EC00843=798156,1112951
EC00844=798156,1112951
EC00845=798156,1112951
EC00846=798156,1112951
EC00847=798156,1112951
EC00848=798156,1112951
EC00849=798156,1112951
EC00850=798156,1112951
EC00851=798156,1112951
EC00852=798156,1112951
EC00853=798156,1112951
EC00854=798156,1112951
EC00855=798156,1112951
EC00856=798156,1112951
EC00857=798156,1112951
EC00858=798156,1112951
EC00859=798156,1112951
EC00860=798156,1112951
EC00861=798156,1112951
EC00862=798156,1112951
EC00863=798156,1112951
EC00864=798156,1112951
EC00865=798156,1112951
EC00866=798156,1112951
EC00867=798156,1112951
EC00868=798156,1112951
EC00869=798156,1112951
EC00870=798156,1112951
EC00871=798156,1112951
EC00872=798156,1112951
EC00873=798156,1112951
EC00874=798156,1112951
EC00875=798156,1112951
EC00876=798156,1112951
EC00877=798156,1112949
EC00878=798156,1112951
EC00879=798156,1112951
EC00880=798156,1112951
EC00881=798156,1112951
EC00882=798156,1112951
EC00883=798156,1112951
EC00884=798156,1112951
EC00885=798156,1112951
EC00886=798156,1112951
EC00887=798156,1112951
EC00888=798156,1112951
EC00889=798156,1112951
EC00890=798156,1112951
EC00891=798156,1112951
EC00892=798156,1112951
EC00893=798156,1112951
EC00894=798156,1112951
EC00895=798156,1112951
EC00896=798156,1112951
EC00897=798156,1112951
EC00898=798156,1112951
EC00899=798156,1112951
EC00900=798156,1112951
EC00901=798156,1112951
EC00902=798156,1112951
EC00903=798156,1112951
EC00904=798156,1112951
EC00905=798156,1112951
EC00906=798156,1112951
EC00907=798156,1112951
EC00908=798156,1112951
EC00909=798156,1112951
EC00910=798156,1112951
EC00911=798156,1112951
EC00912=798156,1112951
EC00913=798156,1112951
EC00914=798156,1112951
EC00915=798156,1112951
EC00916=798156,1112951
EC00917=798156,1112951
EC00918=798156,1112951
EC00919=798156,1112951
EC00920=798156,1112951
EC00921=798156,1112951
EC00922=798156,1112951
EC00923=798156,1112951
EC00924=798156,1112951
EC00925=798156,1112951
EC00926=798156,1112951
EC00927=798156,1112951
EC00928=798156,1112951
EC00929=798156,1112951
EC00930=798156,1112951
EC00931=798156,1112951
EC00932=798156,1112951
EC00933=798156,1112951
EC00934=798156,1112951
EC00935=798156,1112951
EC00936=798156,1112951
EC00937=798156,1112951
EC00938=798156,1112951
EC00939=798156,1112951
EC00940=798156,1112951
EC00941=798156,1112951
EC00942=798155,1112950
EC00943=798155,1112950
EC00944=798155,1112950
EC00945=798155,1112950
EC00946=798155,1112950
EC00947=798155,1112950
EC00948=798155,1112950
EC00949=798156,1112951
EC00950=798156,1112951
EC00951=798156,1112951
EC00952=798156,1112951
EC00953=798156,1112951
EC00954=798156,1112951
EC00955=798156,1112951
EC00956=798156,1112951
EC00957=798156,1112951
EC00958=798156,1112951
EC00959=798156,1112951
EC00960=798156,1112951
EC00961=798156,1112951
EC00962=798156,1112951
EC00963=798156,1112951
EC00964=798156,1112951
EC00965=798156,1112951
EC00966=798156,1112951
EC00967=798156,1112951
EC00968=798156,1112951
EC00969=798156,1112951
EC00970=798156,1112951
EC00971=798156,1112951
EC00972=798156,1112951
EC00973=798156,1112951
EC00974=798156,1112951
EC00975=798156,1112951
EC00976=798156,1112951
EC00977=798156,1112951
EC00978=798156,1112951
EC00979=798156,1112951
EC00980=798156,1112951
EC00981=798156,1112951
EC00982=798156,1112951
EC00983=798156,1112951
EC00984=798156,1112951
EC00985=798156,1112951
EC00986=798156,1112951
EC00987=798156,1112951
EC00988=798156,1112951
EC00989=798156,1112951
EC00990=798156,1112951
EC00991=798156,1112951
EC00992=798156,1112951
EC00993=798156,1112951
EC00994=798156,1112951
EC00995=798156,1112951
EC00996=798156,1112951
EC00997=798156,1112951
EC00998=798156,1112951
EC00999=798156,1112951
EC01000=798156,1112951
EC01001=798156,1112951
EC01002=798156,1112951
EC01003=798156,1112951
EC01004=798156,1112951
EC01005=798156,1112951
EC01006=798156,1112951
EC01007=798156,1112951
EC01008=798156,1112951
EC01009=798156,1112951
EC01010=798156,1112951
EC01011=798156,1112951
EC01012=798156,1112951
EC01013=798156,1112951
EC01014=798156,1112951
EC01015=798156,1112951
EC01016=798155,1112949
EC01017=798156,1112951
EC01018=798156,1112951
EC01019=798156,1112951
EC01020=798156,1112951
EC01021=798156,1112951
EC01022=798156,1112951
EC01023=798156,1112951
EC01024=798156,1112951
EC01025=798156,1112951
EC01026=798156,1112951
EC01027=798156,1112951
EC01028=798156,1112951
EC01029=798156,1112951
EC01030=798156,1112951
EC01031=798156,1112951
EC01032=798156,1112951
EC01033=798156,1112951
EC01034=798156,1112951
///POSTYPE BASE
///RECTAN
///RCONF 0,0,0,0,0,0,0,0,0,0,0,0,0,0,0,0,0,0,0,0,0,0,0,0
P00006=0.222,-3.123,-1.508,0.0000,0.0000,0.0000
P00021=-0.225,-6.128,-0.405,0.0000,0.0000,0.0000
P00022=0.222,-3.123,-1.508,0.0000,0.0000,0.0000
P00023=0.143,-0.036,0.682,0.0000,0.0000,0.0000
P00024=0.145,-0.552,1.326,0.0000,0.0000,0.0000
P00025=-2.003,0.006,0.728,0.0000,0.0000,0.0000
P00026=0.562,-0.002,-0.337,0.0000,0.0000,0.0000
P00027=-0.746,0.015,-9.096,0.0000,0.0000,0.0000
P00028=-2.237,-0.018,-7.702,0.0000,0.0000,0.0000
P00029=-2.156,-0.086,-4.681,0.0000,0.0000,0.0000
P00030=5.926,-4.294,-1.390,0.0000,0.0000,0.0000
P00031=1.853,-0.001,-1.549,0.0000,0.0000,0.0000
P00032=1.957,0.503,-7.217,0.0000,0.0000,0.0000
///RCONF 0,0,0,0,1,0,0,0,0,0,0,0,0,0,0,0,0,0,0,0,0,0,0,0
P00033=-0.123,0.612,-5.012,0.0000,0.0000,0.0000
///RCONF 0,0,0,0,0,0,0,0,0,0,0,0,0,0,0,0,0,0,0,0,0,0,0,0
P00034=-0.304,0.773,-2.693,0.0000,0.0000,0.0000
P00035=2.817,0.591,-1.622,0.0000,0.0000,0.0000
P00040=-0.030,9.648,2.467,0.0000,0.0000,0.0000
P00041=0.192,3.924,0.305,0.0000,0.0000,0.0000
P00042=-0.217,1.941,0.413,0.0000,0.0000,0.0000
P00043=-0.044,-1.937,1.197,0.0000,0.0000,0.0000
P00044=0.687,-2.322,1.156,0.0000,0.0000,0.0000
P00045=-0.068,-0.810,1.603,0.0000,0.0000,0.0000
P00046=0.799,0.043,1.292,0.0000,0.0000,0.0000
///RCONF 0,1,0,0,0,0,0,0,0,0,0,0,0,0,0,0,0,0,0,0,0,0,0,0
P00047=-0.011,1.737,-0.646,0.0000,0.0000,0.0000
///RCONF 0,0,0,0,0,0,0,0,0,0,0,0,0,0,0,0,0,0,0,0,0,0,0,0
P00048=2.411,0.025,-0.606,0.0000,0.0000,0.0000
P00049=3.413,-3.572,-1.618,0.0000,0.0000,0.0000
P00050=4.296,-4.501,-0.826,0.0000,0.0000,0.0000
P00051=0.367,3.892,0.009,0.0000,0.0000,0.0000
P00052=0.088,2.832,-0.342,0.0000,0.0000,0.0000
P00053=0.134,6.594,0.107,0.0000,0.0000,0.0000
P00054=-0.103,6.509,-0.702,0.0000,0.0000,0.0000
P00061=1.575,-3.405,-0.752,0.0000,0.0000,0.0000
P00062=-0.135,-0.848,-1.706,0.0000,0.0000,0.0000
P00063=0.036,-0.654,-3.005,0.0000,0.0000,0.0000
P00071=2.716,0.070,1.352,0.0000,0.0000,0.0000
P00072=1.041,-0.003,-0.797,0.0000,0.0000,0.0000
P00073=-0.961,5.319,-6.157,0.0000,0.0000,0.0000
P00074=1.123,1.944,-5.914,0.0000,0.0000,0.0000
P00080=-3.893,-3.240,-0.208,0.0000,0.0000,0.0000
P00081=19.486,11.347,1.262,0.0000,0.0000,0.0000
P00088=-2.376,0.094,2.453,0.0000,0.0000,0.0000
P00089=5.697,-3.100,-1.263,0.0000,0.0000,0.0000
P00095=-3.945,4.918,-0.177,0.0000,0.0000,0.0000
P00096=-0.633,5.398,-3.809,0.0000,0.0000,0.0000
//INST
///DATE 2024/08/30 11:58
///ATTR SC,RW
///GROUP1 RB1,BS1
///GROUP2 ST1
NOP
'X2_8B-21B(90,180)
'
MOVJ C00000 BC00000 VJ=100.00  +MOVJ EC00000 VJ=100.00
'Path S4722
SFTOF3D
MOVJ C00001 BC00001 VJ=100.00  +MOVJ EC00001 VJ=100.00
MOVL C00002 BC00002 V=666.7  +MOVJ EC00002 VJ=100.00
SMOVL C00003 BC00003 V=166.7  +MOVJ EC00003
SREFP 3 C00004 BC00004  +REFP EC00004
CALL JOB:SEARCH-R1-S13D
SET P095 P006
SFTON3D P095
SMOVL C00005 BC00005 V=166.7  +MOVJ EC00005
SREFP 3 C00006 BC00006  +REFP EC00006
CALL JOB:SEARCH-R1-S13D
SET P095 P006
SFTON3D P095
SMOVL C00007 BC00007 V=166.7  +MOVJ EC00007
MOVL C00008 BC00008 V=1000.0  +MOVJ EC00008 VJ=100.00
'EndPath S4722
'Path S4723
SFTOF3D
MOVJ C00009 BC00009 VJ=100.00  +MOVJ EC00009 VJ=100.00
MOVL C00010 BC00010 V=666.7  +MOVJ EC00010 VJ=100.00
SMOVL C00011 BC00011 V=166.7  +MOVJ EC00011
SREFP 3 C00012 BC00012  +REFP EC00012
CALL JOB:SEARCH-R1-S13D
SET P096 P006
SFTON3D P096
SMOVL C00013 BC00013 V=166.7  +MOVJ EC00013
SREFP 3 C00014 BC00014  +REFP EC00014
CALL JOB:SEARCH-R1-S13D
SET P096 P006
SFTON3D P096
SMOVL C00015 BC00015 V=166.7  +MOVJ EC00015
MOVL C00016 BC00016 V=1000.0  +MOVJ EC00016 VJ=100.00
'EndPath S4723
'
'
'Path S4093
SFTOF3D
MOVJ C00017 BC00017 VJ=100.00  +MOVJ EC00017 VJ=100.00
MOVL C00018 BC00018 V=666.7  +MOVJ EC00018 VJ=100.00
SMOVL C00019 BC00019 V=166.7  +MOVJ EC00019
SREFP 3 C00020 BC00020  +REFP EC00020
CALL JOB:SEARCH-R1-S13D
SET P021 P006
SFTON3D P021
SMOVL C00021 BC00021 V=166.7  +MOVJ EC00021
SREFP 3 C00022 BC00022  +REFP EC00022
CALL JOB:SEARCH-R1-S13D
SET P021 P006
SFTON3D P021
SMOVL C00023 BC00023 V=166.7  +MOVJ EC00023
MOVL C00024 BC00024 V=1000.0  +MOVJ EC00024 VJ=100.00
'EndPath S4093
'Path S4094
SFTOF3D
MOVJ C00025 BC00025 VJ=100.00  +MOVJ EC00025 VJ=100.00
MOVL C00026 BC00026 V=666.7  +MOVJ EC00026 VJ=100.00
SMOVL C00027 BC00027 V=166.7  +MOVJ EC00027
SREFP 3 C00028 BC00028  +REFP EC00028
CALL JOB:SEARCH-R1-S13D
SET P022 P006
SFTON3D P022
SMOVL C00029 BC00029 V=166.7  +MOVJ EC00029
SREFP 3 C00030 BC00030  +REFP EC00030
CALL JOB:SEARCH-R1-S13D
SET P022 P006
SFTON3D P022
SMOVL C00031 BC00031 V=166.7  +MOVJ EC00031
MOVL C00032 BC00032 V=1000.0  +MOVJ EC00032 VJ=100.00
'EndPath S4094
MOVJ C00033 BC00033 VJ=100.00  +MOVJ EC00033 VJ=100.00
'Path S4205
SFTOF3D
MOVJ C00034 BC00034 VJ=100.00  +MOVJ EC00034 VJ=100.00
MOVL C00035 BC00035 V=666.7  +MOVJ EC00035 VJ=100.00
SMOVL C00036 BC00036 V=166.7  +MOVJ EC00036
SREFP 3 C00037 BC00037  +REFP EC00037
CALL JOB:SEARCH-R1-S13D
SET P050 P006
SFTON3D P050
SMOVL C00038 BC00038 V=166.7  +MOVJ EC00038
SREFP 3 C00039 BC00039  +REFP EC00039
CALL JOB:SEARCH-R1-S13D
SET P050 P006
SFTON3D P050
SMOVL C00040 BC00040 V=166.7  +MOVJ EC00040
SMOVL C00041 BC00041 V=250.0  +MOVJ EC00041
SMOVL C00042 BC00042 V=166.7  +MOVJ EC00042
SREFP 3 C00043 BC00043  +REFP EC00043
CALL JOB:SEARCH-R1-S13D
SET P050 P006
SFTON3D P050
SMOVL C00044 BC00044 V=250.0  +MOVJ EC00044
'EndPath S4205
'Path S4206
SFTOF3D
MOVL C00045 BC00045 V=1000.0  +MOVJ EC00045 VJ=100.00
SMOVL C00046 BC00046 V=166.7  +MOVJ EC00046
SREFP 3 C00047 BC00047  +REFP EC00047
CALL JOB:SEARCH-R1-S13D
SET P051 P006
SFTON3D P051
SMOVL C00048 BC00048 V=166.7  +MOVJ EC00048
SREFP 3 C00049 BC00049  +REFP EC00049
CALL JOB:SEARCH-R1-S13D
SET P051 P006
SFTON3D P051
SMOVL C00050 BC00050 V=166.7  +MOVJ EC00050
SMOVL C00051 BC00051 V=250.0  +MOVJ EC00051
SREFP 3 C00052 BC00052  +REFP EC00052
CALL JOB:SEARCH-R1-S13D
SET P051 P006
SFTON3D P051
SMOVL C00053 BC00053 V=250.0  +MOVJ EC00053
MOVL C00054 BC00054 V=1000.0  +MOVJ EC00054 VJ=100.00
'EndPath S4206
MOVJ C00055 BC00055 VJ=100.00  +MOVJ EC00055 VJ=100.00
'Path S4207
SFTOF3D
MOVJ C00056 BC00056 VJ=100.00  +MOVJ EC00056 VJ=100.00
MOVL C00057 BC00057 V=666.7  +MOVJ EC00057 VJ=100.00
SMOVL C00058 BC00058 V=166.7  +MOVJ EC00058
SREFP 3 C00059 BC00059  +REFP EC00059
CALL JOB:SEARCH-R1-S13D
SET P054 P006
SFTON3D P054
SMOVL C00060 BC00060 V=250.0  +MOVJ EC00060
SMOVL C00061 BC00061 V=233.3  +MOVJ EC00061
SMOVL C00062 BC00062 V=166.7  +MOVJ EC00062
SREFP 3 C00063 BC00063  +REFP EC00063
CALL JOB:SEARCH-R1-S13D
SET P054 P006
SFTON3D P054
SMOVL C00064 BC00064 V=166.7  +MOVJ EC00064
SMOVL C00065 BC00065 V=416.7  +MOVJ EC00065
SMOVL C00066 BC00066 V=250.0  +MOVJ EC00066
SREFP 3 C00067 BC00067  +REFP EC00067
CALL JOB:SEARCH-R1-S13D
SET P054 P006
SFTON3D P054
SMOVL C00068 BC00068 V=250.0  +MOVJ EC00068
MOVL C00069 BC00069 V=1000.0  +MOVJ EC00069 VJ=100.00
'EndPath S4207
'Path S4095
SFTOF3D
MOVJ C00070 BC00070 VJ=100.00  +MOVJ EC00070 VJ=100.00
MOVJ C00071 BC00071 VJ=100.00  +MOVJ EC00071 VJ=100.00
SMOVL C00072 BC00072 V=200.0  +MOVJ EC00072
SREFP 3 C00073 BC00073  +REFP EC00073
CALL JOB:SEARCH-R1-S13D
SET P089 P006
SFTON3D P089
SMOVL C00074 BC00074 V=166.7  +MOVJ EC00074
SMOVL C00075 BC00075 V=166.7  +MOVJ EC00075
SREFP 3 C00076 BC00076  +REFP EC00076
CALL JOB:SEARCH-R1-S13D
SET P089 P006
SFTON3D P089
SMOVL C00077 BC00077 V=166.7  +MOVJ EC00077
SMOVL C00078 BC00078 V=166.7  +MOVJ EC00078
SREFP 3 C00079 BC00079  +REFP EC00079
CALL JOB:SEARCH-R1-S13D
SET P089 P006
SFTON3D P089
SMOVL C00080 BC00080 V=166.7  +MOVJ EC00080
SMOVL C00081 BC00081 V=1000.0  +MOVJ EC00081
SFTOF3D
MOVJ C00082 BC00082 VJ=100.00  +MOVJ EC00082 VJ=100.00
MOVL C00083 BC00083 V=666.7  +MOVJ EC00083 VJ=100.00
SMOVL C00084 BC00084 V=166.7  +MOVJ EC00084
SREFP 3 C00085 BC00085  +REFP EC00085
CALL JOB:SEARCH-R1-S13D
SET P034 P006
SFTON3D P034
SMOVL C00086 BC00086 V=250.0  +MOVJ EC00086
SMOVL C00087 BC00087 V=233.3  +MOVJ EC00087
SMOVL C00088 BC00088 V=166.7  +MOVJ EC00088
SREFP 3 C00089 BC00089  +REFP EC00089
CALL JOB:SEARCH-R1-S13D
SET P034 P006
SFTON3D P034
SMOVL C00090 BC00090 V=166.7  +MOVJ EC00090
SMOVL C00091 BC00091 V=166.7  +MOVJ EC00091
SREFP 3 C00092 BC00092  +REFP EC00092
CALL JOB:SEARCH-R1-S13D
SET P034 P006
SFTON3D P034
SMOVL C00093 BC00093 V=166.7  +MOVJ EC00093
MOVJ C00094 BC00094 VJ=50.00  +MOVJ EC00094 VJ=30.00
'EndPath S4095
'Path S4096
SFTOF3D
MOVJ C00095 BC00095 VJ=50.00  +MOVJ EC00095 VJ=30.00
MOVJ C00096 BC00096 VJ=50.00  +MOVJ EC00096 VJ=30.00
MOVJ C00097 BC00097 VJ=50.00  +MOVJ EC00097 VJ=30.00
SMOVL C00098 BC00098 V=166.7  +MOVJ EC00098
SREFP 3 C00099 BC00099  +REFP EC00099
CALL JOB:SEARCH-R1-S13D
SET P061 P006
SFTON3D P061
SMOVL C00100 BC00100 V=166.7  +MOVJ EC00100
SREFP 3 C00101 BC00101  +REFP EC00101
CALL JOB:SEARCH-R1-S13D
SET P061 P006
SFTON3D P061
SMOVL C00102 BC00102 V=166.7  +MOVJ EC00102
SFTOF3D
SMOVL C00103 BC00103 V=666.7  +MOVJ EC00103
SMOVL C00104 BC00104 V=166.7  +MOVJ EC00104
SREFP 3 C00105 BC00105  +REFP EC00105
CALL JOB:SEARCH-R1-S13D
SET P062 P006
SFTON3D P062
SMOVL C00106 BC00106 V=166.7  +MOVJ EC00106
SREFP 3 C00107 BC00107  +REFP EC00107
CALL JOB:SEARCH-R1-S13D
SET P062 P006
SFTON3D P062
SMOVL C00108 BC00108 V=250.0  +MOVJ EC00108
SFTOF3D
SMOVL C00109 BC00109 V=500.0  +MOVJ EC00109
SMOVL C00110 BC00110 V=166.7  +MOVJ EC00110
SREFP 3 C00111 BC00111  +REFP EC00111
CALL JOB:SEARCH-R1-S13D
SET P063 P006
SFTON3D P063
SMOVL C00112 BC00112 V=166.7  +MOVJ EC00112
SREFP 3 C00113 BC00113  +REFP EC00113
CALL JOB:SEARCH-R1-S13D
SET P063 P006
SFTON3D P063
SMOVL C00114 BC00114 V=166.7  +MOVJ EC00114
SFTOF3D
SMOVL C00115 BC00115 V=1000.0  +MOVJ EC00115
MOVJ C00116 BC00116 VJ=100.00  +MOVJ EC00116 VJ=30.00
MOVJ C00117 BC00117 VJ=50.00  +MOVJ EC00117 VJ=30.00
MOVJ C00118 BC00118 VJ=100.00  +MOVJ EC00118 VJ=100.00
MOVL C00119 BC00119 V=666.7  +MOVJ EC00119 VJ=100.00
SMOVL C00120 BC00120 V=166.7  +MOVJ EC00120
SREFP 3 C00121 BC00121  +REFP EC00121
CALL JOB:SEARCH-R1-S13D
SET P023 P006
SFTON3D P023
SMOVL C00122 BC00122 V=166.7  +MOVJ EC00122
SMOVL C00123 BC00123 V=333.3  +MOVJ EC00123
SMOVL C00124 BC00124 V=166.7  +MOVJ EC00124
SREFP 3 C00125 BC00125  +REFP EC00125
CALL JOB:SEARCH-R1-S13D
SET P023 P006
SFTON3D P023
SMOVL C00126 BC00126 V=166.7  +MOVJ EC00126
SMOVL C00127 BC00127 V=166.7  +MOVJ EC00127
SREFP 3 C00128 BC00128  +REFP EC00128
CALL JOB:SEARCH-R1-S13D
SET P023 P006
SFTON3D P023
SMOVL C00129 BC00129 V=166.7  +MOVJ EC00129
MOVL C00130 BC00130 V=1000.0  +MOVJ EC00130 VJ=100.00
'EndPath S4096
MOVJ C00131 BC00131 VJ=100.00  +MOVJ EC00131 VJ=100.00
'Path S4097
SFTOF3D
MOVJ C00132 BC00132 VJ=100.00  +MOVJ EC00132 VJ=100.00
MOVL C00133 BC00133 V=666.7  +MOVJ EC00133 VJ=100.00
SMOVL C00134 BC00134 V=166.7  +MOVJ EC00134
SREFP 3 C00135 BC00135  +REFP EC00135
CALL JOB:SEARCH-R1-S13D
SET P024 P006
SFTON3D P024
SMOVL C00136 BC00136 V=166.7  +MOVJ EC00136
SREFP 3 C00137 BC00137  +REFP EC00137
CALL JOB:SEARCH-R1-S13D
SET P024 P006
SFTON3D P024
SMOVL C00138 BC00138 V=166.7  +MOVJ EC00138
SMOVL C00139 BC00139 V=166.7  +MOVJ EC00139
SREFP 3 C00140 BC00140  +REFP EC00140
CALL JOB:SEARCH-R1-S13D
SET P024 P006
SFTON3D P024
SMOVL C00141 BC00141 V=166.7  +MOVJ EC00141
MOVL C00142 BC00142 V=1000.0  +MOVJ EC00142 VJ=100.00
'EndPath S4097
'Path S4098
SFTOF3D
MOVJ C00143 BC00143 VJ=100.00  +MOVJ EC00143 VJ=100.00
MOVL C00144 BC00144 V=666.7  +MOVJ EC00144 VJ=100.00
SMOVL C00145 BC00145 V=166.7  +MOVJ EC00145
SREFP 3 C00146 BC00146  +REFP EC00146
CALL JOB:SEARCH-R1-S13D
SET P035 P006
SFTON3D P035
SMOVL C00147 BC00147 V=166.7  +MOVJ EC00147
SREFP 3 C00148 BC00148  +REFP EC00148
CALL JOB:SEARCH-R1-S13D
SET P035 P006
SFTON3D P035
SMOVL C00149 BC00149 V=166.7  +MOVJ EC00149
SMOVL C00150 BC00150 V=166.7  +MOVJ EC00150
SMOVL C00151 BC00151 V=166.7  +MOVJ EC00151
SREFP 3 C00152 BC00152  +REFP EC00152
CALL JOB:SEARCH-R1-S13D
SET P035 P006
SFTON3D P035
SMOVL C00153 BC00153 V=166.7  +MOVJ EC00153
MOVL C00154 BC00154 V=1000.0  +MOVJ EC00154 VJ=100.00
'EndPath S4098
'Path S4099
SFTOF3D
MOVJ C00155 BC00155 VJ=100.00  +MOVJ EC00155 VJ=100.00
MOVL C00156 BC00156 V=666.7  +MOVJ EC00156 VJ=100.00
SMOVL C00157 BC00157 V=166.7  +MOVJ EC00157
SREFP 3 C00158 BC00158  +REFP EC00158
CALL JOB:SEARCH-R1-S13D
SET P029 P006
SFTON3D P029
SMOVL C00159 BC00159 V=166.7  +MOVJ EC00159
SREFP 3 C00160 BC00160  +REFP EC00160
CALL JOB:SEARCH-R1-S13D
SET P029 P006
SFTON3D P029
SMOVL C00161 BC00161 V=166.7  +MOVJ EC00161
SMOVL C00162 BC00162 V=250.0  +MOVJ EC00162
SMOVL C00163 BC00163 V=166.7  +MOVJ EC00163
SREFP 3 C00164 BC00164  +REFP EC00164
CALL JOB:SEARCH-R1-S13D
SET P029 P006
SFTON3D P029
SMOVL C00165 BC00165 V=166.7  +MOVJ EC00165
'EndPath S4099
'Path S4855
SFTOF3D
MOVL C00166 BC00166 V=666.7  +MOVJ EC00166 VJ=100.00
SMOVL C00167 BC00167 V=166.7  +MOVJ EC00167
SREFP 3 C00168 BC00168  +REFP EC00168
CALL JOB:SEARCH-R1-S13D
SET P071 P006
SFTON3D P071
SMOVL C00169 BC00169 V=166.7  +MOVJ EC00169
SREFP 3 C00170 BC00170  +REFP EC00170
CALL JOB:SEARCH-R1-S13D
SET P071 P006
SFTON3D P071
SMOVL C00171 BC00171 V=166.7  +MOVJ EC00171
SMOVL C00172 BC00172 V=166.7  +MOVJ EC00172
SREFP 3 C00173 BC00173  +REFP EC00173
CALL JOB:SEARCH-R1-S13D
SET P071 P006
SFTON3D P071
SMOVL C00174 BC00174 V=166.7  +MOVJ EC00174
MOVL C00175 BC00175 V=1000.0  +MOVJ EC00175 VJ=100.00
MOVL C00176 BC00176 V=666.7  +MOVJ EC00176 VJ=100.00
SMOVL C00177 BC00177 V=166.7  +MOVJ EC00177
SREFP 3 C00178 BC00178  +REFP EC00178
CALL JOB:SEARCH-R1-S13D
SET P080 P006
SFTON3D P080
SMOVL C00179 BC00179 V=166.7  +MOVJ EC00179
SREFP 3 C00180 BC00180  +REFP EC00180
CALL JOB:SEARCH-R1-S13D
SET P080 P006
SFTON3D P080
SMOVL C00181 BC00181 V=166.7  +MOVJ EC00181
SMOVL C00182 BC00182 V=250.0  +MOVJ EC00182
SMOVL C00183 BC00183 V=166.7  +MOVJ EC00183
SREFP 3 C00184 BC00184  +REFP EC00184
CALL JOB:SEARCH-R1-S13D
SET P080 P006
SFTON3D P080
SMOVL C00185 BC00185 V=166.7  +MOVJ EC00185
'EndPath S4855
'Path S4856
SFTOF3D
MOVJ C00186 BC00186 VJ=100.00  +MOVJ EC00186 VJ=100.00
MOVL C00187 BC00187 V=666.7  +MOVJ EC00187 VJ=100.00
SMOVL C00188 BC00188 V=166.7  +MOVJ EC00188
SREFP 3 C00189 BC00189  +REFP EC00189
CALL JOB:SEARCH-R1-S13D
SET P072 P006
SFTON3D P072
SMOVL C00190 BC00190 V=166.7  +MOVJ EC00190
SREFP 3 C00191 BC00191  +REFP EC00191
CALL JOB:SEARCH-R1-S13D
SET P072 P006
SFTON3D P072
SMOVL C00192 BC00192 V=166.7  +MOVJ EC00192
MOVL C00193 BC00193 V=1000.0  +MOVJ EC00193 VJ=100.00
'EndPath S4856
MOVJ C00194 BC00194 VJ=100.00  +MOVJ EC00194 VJ=100.00
'Path S4857
SFTOF3D
MOVJ C00195 BC00195 VJ=100.00  +MOVJ EC00195 VJ=100.00
MOVL C00196 BC00196 V=666.7  +MOVJ EC00196 VJ=100.00
SMOVL C00197 BC00197 V=166.7  +MOVJ EC00197
SREFP 3 C00198 BC00198  +REFP EC00198
CALL JOB:SEARCH-R1-S13D
SET P073 P006
SFTON3D P073
SMOVL C00199 BC00199 V=166.7  +MOVJ EC00199
SMOVL C00200 BC00200 V=166.7  +MOVJ EC00200
SREFP 3 C00201 BC00201  +REFP EC00201
CALL JOB:SEARCH-R1-S13D
SET P073 P006
SFTON3D P073
SMOVL C00202 BC00202 V=166.7  +MOVJ EC00202
SMOVL C00203 BC00203 V=166.7  +MOVJ EC00203
SREFP 3 C00204 BC00204  +REFP EC00204
CALL JOB:SEARCH-R1-S13D
SET P073 P006
SFTON3D P073
SMOVL C00205 BC00205 V=166.7  +MOVJ EC00205
MOVL C00206 BC00206 V=1000.0  +MOVJ EC00206 VJ=100.00
'EndPath S4857
MOVJ C00207 BC00207 VJ=100.00  +MOVJ EC00207 VJ=100.00
MOVJ C00208 BC00208 VJ=100.00  +MOVJ EC00208 VJ=100.00
'Path S4858
SFTOF3D
MOVJ C00209 BC00209 VJ=100.00  +MOVJ EC00209 VJ=100.00
MOVL C00210 BC00210 V=666.7  +MOVJ EC00210 VJ=100.00
SMOVL C00211 BC00211 V=166.7  +MOVJ EC00211
SREFP 3 C00212 BC00212  +REFP EC00212
CALL JOB:SEARCH-R1-S13D
SET P074 P006
SFTON3D P074
SMOVL C00213 BC00213 V=166.7  +MOVJ EC00213
SREFP 3 C00214 BC00214  +REFP EC00214
CALL JOB:SEARCH-R1-S13D
SET P074 P006
SFTON3D P074
SMOVL C00215 BC00215 V=166.7  +MOVJ EC00215
MOVL C00216 BC00216 V=1000.0  +MOVJ EC00216 VJ=100.00
'EndPath S4858
MOVJ C00217 BC00217 VJ=100.00  +MOVJ EC00217 VJ=100.00
MOVJ C00218 BC00218 VJ=100.00  +MOVJ EC00218 VJ=100.00
'Path S4100
SFTOF3D
MOVJ C00219 BC00219 VJ=100.00  +MOVJ EC00219 VJ=100.00
MOVL C00220 BC00220 V=666.7  +MOVJ EC00220 VJ=100.00
SMOVL C00221 BC00221 V=166.7  +MOVJ EC00221
SREFP 3 C00222 BC00222  +REFP EC00222
CALL JOB:SEARCH-R1-S13D
SET P081 P006
SFTON3D P081
SMOVL C00223 BC00223 V=166.7  +MOVJ EC00223
SREFP 3 C00224 BC00224  +REFP EC00224
CALL JOB:SEARCH-R1-S13D
SET P081 P006
SFTON3D P081
SMOVL C00225 BC00225 V=166.7  +MOVJ EC00225
SMOVL C00226 BC00226 V=666.7  +MOVJ EC00226
SMOVL C00227 BC00227 V=666.7  +MOVJ EC00227
SMOVL C00228 BC00228 V=666.7  +MOVJ EC00228
SMOVL C00229 BC00229 V=166.7  +MOVJ EC00229
SREFP 3 C00230 BC00230  +REFP EC00230
CALL JOB:SEARCH-R1-S13D
SET P081 P006
SFTON3D P081
SMOVL C00231 BC00231 V=250.0  +MOVJ EC00231
SMOVL C00232 BC00232 V=666.7  +MOVJ EC00232
MOVJ C00233 BC00233 VJ=100.00  +MOVJ EC00233 VJ=100.00
MOVL C00234 BC00234 V=666.7  +MOVJ EC00234 VJ=100.00
SMOVL C00235 BC00235 V=166.7  +MOVJ EC00235
SREFP 3 C00236 BC00236  +REFP EC00236
CALL JOB:SEARCH-R1-S13D
SET P026 P006
SFTON3D P026
SMOVL C00237 BC00237 V=166.7  +MOVJ EC00237
SREFP 3 C00238 BC00238  +REFP EC00238
CALL JOB:SEARCH-R1-S13D
SET P026 P006
SFTON3D P026
SMOVL C00239 BC00239 V=166.7  +MOVJ EC00239
SMOVL C00240 BC00240 V=666.7  +MOVJ EC00240
SMOVL C00241 BC00241 V=666.7  +MOVJ EC00241
SMOVL C00242 BC00242 V=666.7  +MOVJ EC00242
SMOVL C00243 BC00243 V=166.7  +MOVJ EC00243
SREFP 3 C00244 BC00244  +REFP EC00244
CALL JOB:SEARCH-R1-S13D
SET P026 P006
SFTON3D P026
SMOVL C00245 BC00245 V=250.0  +MOVJ EC00245
SMOVL C00246 BC00246 V=666.7  +MOVJ EC00246
MOVL C00247 BC00247 V=1000.0  +MOVJ EC00247 VJ=100.00
'EndPath S4100
MOVJ C00248 BC00248 VJ=50.00  +MOVJ EC00248 VJ=100.00
'Path S4101
SFTOF3D
MOVJ C00249 BC00249 VJ=50.00  +MOVJ EC00249 VJ=100.00
MOVL C00250 BC00250 V=666.7  +MOVJ EC00250 VJ=100.00
SMOVL C00251 BC00251 V=166.7  +MOVJ EC00251
SREFP 3 C00252 BC00252  +REFP EC00252
CALL JOB:SEARCH-R1-S13D
SET P025 P006
SFTON3D P025
SMOVL C00253 BC00253 V=166.7  +MOVJ EC00253
SREFP 3 C00254 BC00254  +REFP EC00254
CALL JOB:SEARCH-R1-S13D
SET P025 P006
SFTON3D P025
SMOVL C00255 BC00255 V=166.7  +MOVJ EC00255
SMOVL C00256 BC00256 V=333.3  +MOVJ EC00256
SMOVL C00257 BC00257 V=166.7  +MOVJ EC00257
SREFP 3 C00258 BC00258  +REFP EC00258
CALL JOB:SEARCH-R1-S13D
SET P025 P006
SFTON3D P025
SMOVL C00259 BC00259 V=166.7  +MOVJ EC00259
MOVL C00260 BC00260 V=1000.0  +MOVJ EC00260 VJ=100.00
'EndPath S4101
MOVJ C00261 BC00261 VJ=100.00  +MOVJ EC00261 VJ=100.00
'Path S4102
SFTOF3D
MOVJ C00262 BC00262 VJ=100.00  +MOVJ EC00262 VJ=100.00
MOVL C00263 BC00263 V=666.7  +MOVJ EC00263 VJ=100.00
SMOVL C00264 BC00264 V=166.7  +MOVJ EC00264
SREFP 3 C00265 BC00265  +REFP EC00265
CALL JOB:SEARCH-R1-S13D
SET P028 P006
SFTON3D P028
SMOVL C00266 BC00266 V=166.7  +MOVJ EC00266
SREFP 3 C00267 BC00267  +REFP EC00267
CALL JOB:SEARCH-R1-S13D
SET P028 P006
SFTON3D P028
SMOVL C00268 BC00268 V=166.7  +MOVJ EC00268
SMOVL C00269 BC00269 V=333.3  +MOVJ EC00269
SMOVL C00270 BC00270 V=166.7  +MOVJ EC00270
SREFP 3 C00271 BC00271  +REFP EC00271
CALL JOB:SEARCH-R1-S13D
SET P028 P006
SFTON3D P028
SMOVL C00272 BC00272 V=166.7  +MOVJ EC00272
MOVL C00273 BC00273 V=1000.0  +MOVJ EC00273 VJ=100.00
'EndPath S4102
MOVJ C00274 BC00274 VJ=100.00  +MOVJ EC00274 VJ=100.00
'Path S4103
SFTOF3D
MOVJ C00275 BC00275 VJ=100.00  +MOVJ EC00275 VJ=100.00
MOVL C00276 BC00276 V=666.7  +MOVJ EC00276 VJ=100.00
SMOVL C00277 BC00277 V=166.7  +MOVJ EC00277
SREFP 3 C00278 BC00278  +REFP EC00278
CALL JOB:SEARCH-R1-S13D
SET P033 P006
SFTON3D P033
SMOVL C00279 BC00279 V=166.7  +MOVJ EC00279
SMOVL C00280 BC00280 V=166.7  +MOVJ EC00280
SREFP 3 C00281 BC00281  +REFP EC00281
CALL JOB:SEARCH-R1-S13D
SET P033 P006
SFTON3D P033
SMOVL C00282 BC00282 V=166.7  +MOVJ EC00282
SMOVL C00283 BC00283 V=166.7  +MOVJ EC00283
SMOVL C00284 BC00284 V=166.7  +MOVJ EC00284
SREFP 3 C00285 BC00285  +REFP EC00285
CALL JOB:SEARCH-R1-S13D
SET P033 P006
SFTON3D P033
SMOVL C00286 BC00286 V=166.7  +MOVJ EC00286
MOVL C00287 BC00287 V=1000.0  +MOVJ EC00287 VJ=100.00
'EndPath S4103
'Path S4104
SFTOF3D
MOVJ C00288 BC00288 VJ=100.00  +MOVJ EC00288 VJ=100.00
MOVL C00289 BC00289 V=666.7  +MOVJ EC00289 VJ=100.00
SMOVL C00290 BC00290 V=166.7  +MOVJ EC00290
SREFP 3 C00291 BC00291  +REFP EC00291
CALL JOB:SEARCH-R1-S13D
SET P027 P006
SFTON3D P027
SMOVL C00292 BC00292 V=250.0  +MOVJ EC00292
SMOVL C00293 BC00293 V=166.7  +MOVJ EC00293
SREFP 3 C00294 BC00294  +REFP EC00294
CALL JOB:SEARCH-R1-S13D
SET P027 P006
SFTON3D P027
SMOVL C00295 BC00295 V=166.7  +MOVJ EC00295
SMOVL C00296 BC00296 V=166.7  +MOVJ EC00296
SREFP 3 C00297 BC00297  +REFP EC00297
CALL JOB:SEARCH-R1-S13D
SET P027 P006
SFTON3D P027
SMOVL C00298 BC00298 V=166.7  +MOVJ EC00298
MOVL C00299 BC00299 V=1000.0  +MOVJ EC00299 VJ=100.00
'EndPath S4104
MOVJ C00300 BC00300 VJ=100.00  +MOVJ EC00300 VJ=100.00
'Path S4105
SFTOF3D
MOVJ C00301 BC00301 VJ=100.00  +MOVJ EC00301 VJ=100.00
MOVL C00302 BC00302 V=666.7  +MOVJ EC00302 VJ=100.00
SMOVL C00303 BC00303 V=166.7  +MOVJ EC00303
SREFP 3 C00304 BC00304  +REFP EC00304
CALL JOB:SEARCH-R1-S13D
SET P030 P006
SFTON3D P030
SMOVL C00305 BC00305 V=166.7  +MOVJ EC00305
SREFP 3 C00306 BC00306  +REFP EC00306
CALL JOB:SEARCH-R1-S13D
SET P030 P006
SFTON3D P030
SMOVL C00307 BC00307 V=166.7  +MOVJ EC00307
MOVL C00308 BC00308 V=1000.0  +MOVJ EC00308 VJ=100.00
'EndPath S4105
'Path S4106
SFTOF3D
MOVJ C00309 BC00309 VJ=100.00  +MOVJ EC00309 VJ=100.00
MOVL C00310 BC00310 V=666.7  +MOVJ EC00310 VJ=100.00
SMOVL C00311 BC00311 V=166.7  +MOVJ EC00311
SREFP 3 C00312 BC00312  +REFP EC00312
CALL JOB:SEARCH-R1-S13D
SET P031 P006
SFTON3D P031
SMOVL C00313 BC00313 V=166.7  +MOVJ EC00313
SREFP 3 C00314 BC00314  +REFP EC00314
CALL JOB:SEARCH-R1-S13D
SET P031 P006
SFTON3D P031
SMOVL C00315 BC00315 V=166.7  +MOVJ EC00315
MOVL C00316 BC00316 V=1000.0  +MOVJ EC00316 VJ=100.00
'EndPath S4106
MOVJ C00317 BC00317 VJ=100.00  +MOVJ EC00317 VJ=100.00
'Path S4107
SFTOF3D
MOVJ C00318 BC00318 VJ=100.00  +MOVJ EC00318 VJ=100.00
MOVL C00319 BC00319 V=666.7  +MOVJ EC00319 VJ=100.00
SMOVL C00320 BC00320 V=166.7  +MOVJ EC00320
SREFP 3 C00321 BC00321  +REFP EC00321
CALL JOB:SEARCH-R1-S13D
SET P032 P006
SFTON3D P032
SMOVL C00322 BC00322 V=166.7  +MOVJ EC00322
SREFP 3 C00323 BC00323  +REFP EC00323
CALL JOB:SEARCH-R1-S13D
SET P032 P006
SFTON3D P032
SMOVL C00324 BC00324 V=166.7  +MOVJ EC00324
SMOVL C00325 BC00325 V=250.0  +MOVJ EC00325
SMOVL C00326 BC00326 V=166.7  +MOVJ EC00326
SREFP 3 C00327 BC00327  +REFP EC00327
CALL JOB:SEARCH-R1-S13D
SET P032 P006
SFTON3D P032
SMOVL C00328 BC00328 V=166.7  +MOVJ EC00328
MOVL C00329 BC00329 V=1000.0  +MOVJ EC00329 VJ=100.00
'EndPath S4107
'
MOVJ C00330 BC00330 VJ=100.00  +MOVJ EC00330 VJ=100.00
'Path S4208
SFTOF3D
MOVJ C00331 BC00331 VJ=100.00  +MOVJ EC00331 VJ=100.00
MOVL C00332 BC00332 V=666.7  +MOVJ EC00332 VJ=100.00
SMOVL C00333 BC00333 V=166.7  +MOVJ EC00333
SREFP 3 C00334 BC00334  +REFP EC00334
CALL JOB:SEARCH-R1-S13D
SET P052 P006
SFTON3D P052
SMOVL C00335 BC00335 V=166.7  +MOVJ EC00335
SREFP 3 C00336 BC00336  +REFP EC00336
CALL JOB:SEARCH-R1-S13D
SET P052 P006
SFTON3D P052
SMOVL C00337 BC00337 V=166.7  +MOVJ EC00337
SFTOF3D
MOVL C00338 BC00338 V=1000.0  +MOVJ EC00338 VJ=100.00
SMOVL C00339 BC00339 V=500.0  +MOVJ EC00339
SMOVL C00340 BC00340 V=166.7  +MOVJ EC00340
SREFP 3 C00341 BC00341  +REFP EC00341
CALL JOB:SEARCH-R1-S13D
SET P088 P006
SFTON3D P088
SMOVL C00342 BC00342 V=166.7  +MOVJ EC00342
SMOVL C00343 BC00343 V=166.7  +MOVJ EC00343
SMOVL C00344 BC00344 V=166.7  +MOVJ EC00344
SREFP 3 C00345 BC00345  +REFP EC00345
CALL JOB:SEARCH-R1-S13D
SET P088 P006
SFTON3D P088
SMOVL C00346 BC00346 V=333.3  +MOVJ EC00346
SMOVL C00347 BC00347 V=666.7  +MOVJ EC00347
SFTOF3D
'EndPath S4208
MOVJ C00348 BC00348 VJ=100.00  +MOVJ EC00348 VJ=100.00
'Path S4209
SFTOF3D
MOVJ C00349 BC00349 VJ=100.00  +MOVJ EC00349 VJ=100.00
MOVL C00350 BC00350 V=666.7  +MOVJ EC00350 VJ=100.00
SMOVL C00351 BC00351 V=166.7  +MOVJ EC00351
SREFP 3 C00352 BC00352  +REFP EC00352
CALL JOB:SEARCH-R1-S13D
SET P053 P006
SFTON3D P053
SMOVL C00353 BC00353 V=166.7  +MOVJ EC00353
SMOVL C00354 BC00354 V=166.7  +MOVJ EC00354
SREFP 3 C00355 BC00355  +REFP EC00355
CALL JOB:SEARCH-R1-S13D
SET P053 P006
SFTON3D P053
SMOVL C00356 BC00356 V=166.7  +MOVJ EC00356
MOVL C00357 BC00357 V=1000.0  +MOVJ EC00357 VJ=100.00
'EndPath S4209
*BP1
MOVJ C00358 BC00358 VJ=100.00  +MOVJ EC00358 VJ=100.00
'Path W4108
SFTOF3D
SFTON3D P033
MOVJ C00359 BC00359 VJ=100.00  +MOVJ EC00359 VJ=100.00
SMOVL C00360 BC00360 V=666.7  +MOVJ EC00360
SMOVL C00361 BC00361 V=166.7 PL=0  +MOVJ EC00361
MACRO1 MJ#(0) ARGF14
ARCON
SMOVL C00362 BC00362 V=9.2  +MOVJ EC00362
ARCOF
SMOVL C00363 BC00363 V=800.0  +MOVJ EC00363
SMOVL C00364 BC00364 V=1000.0  +MOVJ EC00364
SFTOF3D
'EndPath W4108
'Path W4109
SFTOF3D
MOVJ C00365 BC00365 VJ=100.00  +MOVJ EC00365 VJ=100.00
MOVJ C00366 BC00366 VJ=100.00  +MOVJ EC00366 VJ=100.00
'Path W4110
SFTOF3D
SFTON3D P033
MOVJ C00367 BC00367 VJ=100.00  +MOVJ EC00367 VJ=100.00
SMOVL C00368 BC00368 V=800.0  +MOVJ EC00368
SMOVL C00369 BC00369 V=133.3 PL=0  +MOVJ EC00369
MACRO1 MJ#(0) ARGF9
ARCON
SMOVL C00370 BC00370 V=11.7  +MOVJ EC00370
SMOVL C00371 BC00371 V=11.7  +MOVJ EC00371
SMOVL C00372 BC00372 V=11.7  +MOVJ EC00372
ARCOF
SMOVL C00373 BC00373 V=800.0  +MOVJ EC00373
SMOVL C00374 BC00374 V=1000.0  +MOVJ EC00374
SFTOF3D
'EndPath W4110
MOVJ C00375 BC00375 VJ=100.00  +MOVJ EC00375 VJ=100.00
'9
MOVJ C00376 BC00376 VJ=100.00  +MOVJ EC00376 VJ=100.00
'Path W4111
SFTOF3D
SFTON3D P026
MOVJ C00377 BC00377 VJ=100.00  +MOVJ EC00377 VJ=100.00
SMOVL C00378 BC00378 V=666.7  +MOVJ EC00378
SMOVL C00379 BC00379 V=166.7 PL=0  +MOVJ EC00379
MACRO1 MJ#(0) ARGF14
ARCON
SMOVL C00380 BC00380 V=9.2  +MOVJ EC00380
ARCOF
SMOVL C00381 BC00381 V=800.0  +MOVJ EC00381
SMOVL C00382 BC00382 V=1000.0  +MOVJ EC00382
SFTOF3D
'EndPath W4111
'Path W4112
SFTOF3D
SFTON3D P026
MOVJ C00383 BC00383 VJ=100.00  +MOVJ EC00383 VJ=100.00
SMOVL C00384 BC00384 V=800.0  +MOVJ EC00384
SMOVL C00385 BC00385 V=150.0 PL=0  +MOVJ EC00385
ARCON
SMOVL C00386 BC00386 V=11.7  +MOVJ EC00386
SMOVL C00387 BC00387 V=11.7  +MOVJ EC00387
SMOVL C00388 BC00388 V=11.7  +MOVJ EC00388
ARCOF
SMOVL C00389 BC00389 V=800.0  +MOVJ EC00389
SMOVL C00390 BC00390 V=1000.0  +MOVJ EC00390
SFTOF3D
MOVJ C00391 BC00391 VJ=100.00  +MOVJ EC00391 VJ=100.00
MOVJ C00392 BC00392 VJ=100.00  +MOVJ EC00392 VJ=100.00
'uwaga na podajnik
'Path W4114
SFTOF3D
SFTON3D P026
MOVJ C00393 BC00393 VJ=100.00  +MOVJ EC00393 VJ=100.00
SMOVL C00394 BC00394 V=800.0  +MOVJ EC00394
SMOVL C00395 BC00395 V=150.0 PL=0  +MOVJ EC00395
ARCON
SMOVL C00396 BC00396 V=11.7  +MOVJ EC00396
ARCOF
SMOVL C00397 BC00397 V=800.0  +MOVJ EC00397
SMOVL C00398 BC00398 V=1000.0  +MOVJ EC00398
SFTOF3D
'EndPath W4114
'brak dostepu offset drutu 1cm
'Path W4115
SFTOF3D
SFTON3D P026
MOVJ C00399 BC00399 VJ=100.00  +MOVJ EC00399 VJ=100.00
SMOVL C00400 BC00400 V=800.0  +MOVJ EC00400
SMOVL C00401 BC00401 V=150.0 PL=0  +MOVJ EC00401
ARCON
SMOVL C00402 BC00402 V=11.7  +MOVJ EC00402
ARCOF
SMOVL C00403 BC00403 V=800.0  +MOVJ EC00403
SMOVL C00404 BC00404 V=1000.0  +MOVJ EC00404
SFTOF3D
SFTON3D P081
MOVJ C00405 BC00405 VJ=100.00  +MOVJ EC00405 VJ=100.00
SMOVL C00406 BC00406 V=666.7  +MOVJ EC00406
SMOVL C00407 BC00407 V=166.7 PL=0  +MOVJ EC00407
MACRO1 MJ#(0) ARGF14
ARCON
SMOVL C00408 BC00408 V=9.2  +MOVJ EC00408
ARCOF
SMOVL C00409 BC00409 V=800.0  +MOVJ EC00409
SMOVL C00410 BC00410 V=1000.0  +MOVJ EC00410
SFTOF3D
'EndPath W4111
'Path W4112
SFTOF3D
SFTON3D P081
MOVJ C00411 BC00411 VJ=100.00  +MOVJ EC00411 VJ=100.00
SMOVL C00412 BC00412 V=800.0  +MOVJ EC00412
SMOVL C00413 BC00413 V=150.0 PL=0  +MOVJ EC00413
ARCON
SMOVL C00414 BC00414 V=11.7  +MOVJ EC00414
SMOVL C00415 BC00415 V=11.7  +MOVJ EC00415
SMOVL C00416 BC00416 V=11.7  +MOVJ EC00416
ARCOF
SMOVL C00417 BC00417 V=800.0  +MOVJ EC00417
SMOVL C00418 BC00418 V=1000.0  +MOVJ EC00418
SFTOF3D
MOVJ C00419 BC00419 VJ=100.00  +MOVJ EC00419 VJ=100.00
MOVJ C00420 BC00420 VJ=100.00  +MOVJ EC00420 VJ=100.00
'uwaga na podajnik
'Path W4114
SFTOF3D
SFTON3D P081
MOVJ C00421 BC00421 VJ=100.00  +MOVJ EC00421 VJ=100.00
SMOVL C00422 BC00422 V=800.0  +MOVJ EC00422
SMOVL C00423 BC00423 V=150.0 PL=0  +MOVJ EC00423
ARCON
SMOVL C00424 BC00424 V=11.7  +MOVJ EC00424
ARCOF
SMOVL C00425 BC00425 V=800.0  +MOVJ EC00425
SMOVL C00426 BC00426 V=1000.0  +MOVJ EC00426
SFTOF3D
'EndPath W4114
'brak dostepu offset drutu 1cm
'Path W4115
SFTOF3D
SFTON3D P081
MOVJ C00427 BC00427 VJ=100.00  +MOVJ EC00427 VJ=100.00
SMOVL C00428 BC00428 V=800.0  +MOVJ EC00428
SMOVL C00429 BC00429 V=150.0 PL=0  +MOVJ EC00429
ARCON
SMOVL C00430 BC00430 V=11.7  +MOVJ EC00430
ARCOF
SMOVL C00431 BC00431 V=800.0  +MOVJ EC00431
SMOVL C00432 BC00432 V=1000.0  +MOVJ EC00432
SFTOF3D
'EndPath W4115
MOVJ C00433 BC00433 VJ=100.00  +MOVJ EC00433 VJ=100.00
'10
'11
MOVJ C00434 BC00434 VJ=100.00  +MOVJ EC00434 VJ=100.00
'Path W4118
SFTOF3D
SFTON3D P025
MOVJ C00435 BC00435 VJ=100.00  +MOVJ EC00435 VJ=100.00
SMOVL C00436 BC00436 V=800.0  +MOVJ EC00436
SMOVL C00437 BC00437 V=166.7  +MOVJ EC00437
ARCON
SMOVL C00438 BC00438 V=9.2  +MOVJ EC00438
SMOVL C00439 BC00439 V=9.2  +MOVJ EC00439
SMOVL C00440 BC00440 V=9.2  +MOVJ EC00440
SMOVL C00441 BC00441 V=9.2  +MOVJ EC00441
SMOVL C00442 BC00442 V=9.2  +MOVJ EC00442
ARCOF
SMOVL C00443 BC00443 V=800.0  +MOVJ EC00443
SMOVL C00444 BC00444 V=1000.0  +MOVJ EC00444
SFTOF3D
'EndPath W4118
'brak dostepu offset drutu 1cm
MOVJ C00445 BC00445 VJ=100.00  +MOVJ EC00445 VJ=100.00
'Path W4117
SFTOF3D
SFTON3D P025
MOVJ C00446 BC00446 VJ=100.00  +MOVJ EC00446 VJ=100.00
SMOVL C00447 BC00447 V=800.0  +MOVJ EC00447
SMOVL C00448 BC00448 V=166.7 PL=0  +MOVJ EC00448
ARCON
SMOVL C00449 BC00449 V=10.0  +MOVJ EC00449
ARCOF
SMOVL C00450 BC00450 V=800.0  +MOVJ EC00450
SMOVL C00451 BC00451 V=1000.0  +MOVJ EC00451
SFTOF3D
'EndPath W4117
'12
MOVJ C00452 BC00452 VJ=100.00  +MOVJ EC00452 VJ=100.00
MOVJ C00453 BC00453 VJ=100.00  +MOVJ EC00453 VJ=100.00
'Path W4859
SFTOF3D
SFTON3D P073
MOVJ C00454 BC00454 VJ=100.00  +MOVJ EC00454 VJ=100.00
SMOVL C00455 BC00455 V=800.0  +MOVJ EC00455
SMOVL C00456 BC00456 V=150.0 PL=0  +MOVJ EC00456
ARCON
SMOVL C00457 BC00457 V=8.3  +MOVJ EC00457
SFTON3D P074
SMOVL C00458 BC00458 V=9.2  +MOVJ EC00458
ARCOF
SMOVL C00459 BC00459 V=333.3  +MOVJ EC00459
SMOVL C00460 BC00460 V=333.3  +MOVJ EC00460
SMOVL C00461 BC00461 V=333.3  +MOVJ EC00461
SMOVL C00462 BC00462 V=166.7 PL=0  +MOVJ EC00462
ARCON
SMOVL C00463 BC00463 V=9.2  +MOVJ EC00463
SMOVL C00464 BC00464 V=9.2  +MOVJ EC00464
ARCOF
SMOVL C00465 BC00465 V=800.0  +MOVJ EC00465
SMOVL C00466 BC00466 V=1000.0  +MOVJ EC00466
SFTOF3D
'EndPath W4859
MOVJ C00467 BC00467 VJ=100.00  +MOVJ EC00467 VJ=100.00
MOVJ C00468 BC00468 VJ=100.00  +MOVJ EC00468 VJ=100.00
'Path W4119
SFTOF3D
SFTON3D P034
MOVJ C00469 BC00469 VJ=100.00  +MOVJ EC00469 VJ=100.00
SMOVL C00470 BC00470 V=800.0  +MOVJ EC00470
SMOVL C00471 BC00471 V=150.0 PL=0  +MOVJ EC00471
ARCON
SMOVL C00472 BC00472 V=10.0  +MOVJ EC00472
SMOVL C00473 BC00473 V=10.0  +MOVJ EC00473
SMOVL C00474 BC00474 V=10.0  +MOVJ EC00474
ARCOF
SMOVL C00475 BC00475 V=800.0  +MOVJ EC00475
SMOVL C00476 BC00476 V=1000.0  +MOVJ EC00476
SFTOF3D
'EndPath W4119
'Path W4210
SFTOF3D
SFTON3D P050
MOVJ C00477 BC00477 VJ=100.00  +MOVJ EC00477 VJ=100.00
SMOVL C00478 BC00478 V=800.0  +MOVJ EC00478
SMOVL C00479 BC00479 V=150.0 PL=0  +MOVJ EC00479
ARCON
SMOVL C00480 BC00480 V=11.7  +MOVJ EC00480
ARCOF
SMOVL C00481 BC00481 V=800.0  +MOVJ EC00481
SMOVL C00482 BC00482 V=1000.0  +MOVJ EC00482
SFTOF3D
'EndPath W4210
'Path W4211
SFTOF3D
SFTON3D P034
MOVJ C00483 BC00483 VJ=100.00  +MOVJ EC00483 VJ=100.00
SMOVL C00484 BC00484 V=800.0  +MOVJ EC00484
SMOVL C00485 BC00485 V=166.7 PL=0  +MOVJ EC00485
ARCON
SWVON WEV#(66)
SMOVL C00486 BC00486 V=9.2  +MOVJ EC00486
SMOVL C00487 BC00487 V=9.2  +MOVJ EC00487
SMOVL C00488 BC00488 V=9.2  +MOVJ EC00488
ARCOF
SMOVL C00489 BC00489 V=800.0  +MOVJ EC00489
SMOVL C00490 BC00490 V=1000.0  +MOVJ EC00490
MOVJ C00491 BC00491 VJ=30.00  +MOVJ EC00491 VJ=30.00
MOVJ C00492 BC00492 VJ=30.00  +MOVJ EC00492 VJ=30.00
SFTOF3D
MACRO1 MJ#(0) ARGF6
MOVJ C00493 BC00493 VJ=30.00  +MOVJ EC00493 VJ=30.00
SFTON3D P063
SMOVL C00494 BC00494 V=133.3  +MOVJ EC00494
ARCON
SMOVL C00495 BC00495 V=11.7  +MOVJ EC00495
SMOVL C00496 BC00496 V=11.7  +MOVJ EC00496
SMOVL C00497 BC00497 V=11.7  +MOVJ EC00497
SFTON3D P062
SMOVL C00498 BC00498 V=11.7  +MOVJ EC00498
SMOVL C00499 BC00499 V=11.7  +MOVJ EC00499
SFTON3D P061
SMOVL C00500 BC00500 V=11.0  +MOVJ EC00500
SMOVL C00501 BC00501 V=11.0  +MOVJ EC00501
ARCOF
SMOVL C00502 BC00502 V=250.0  +MOVJ EC00502
SFTOF3D
MOVJ C00503 BC00503 VJ=30.00  +MOVJ EC00503 VJ=30.00
MOVJ C00504 BC00504 VJ=30.00  +MOVJ EC00504 VJ=30.00
'EndPath W4211
'Path W4210
SFTOF3D
SFTON3D P054
MOVJ C00505 BC00505 VJ=100.00  +MOVJ EC00505 VJ=100.00
SMOVL C00506 BC00506 V=800.0  +MOVJ EC00506
SMOVL C00507 BC00507 V=150.0 PL=0  +MOVJ EC00507
MACRO1 MJ#(0) ARGF14
ARCON
SWVON WEV#(67)
SMOVL C00508 BC00508 V=10.0  +MOVJ EC00508
SMOVL C00509 BC00509 V=10.0  +MOVJ EC00509
ARCOF
SWVOF
SMOVL C00510 BC00510 V=800.0  +MOVJ EC00510
SMOVL C00511 BC00511 V=1000.0  +MOVJ EC00511
SFTOF3D
'EndPath W4210
'Path W4121
SFTOF3D
SFTON3D P028
MOVJ C00512 BC00512 VJ=100.00  +MOVJ EC00512 VJ=100.00
SMOVL C00513 BC00513 V=800.0  +MOVJ EC00513
SMOVL C00514 BC00514 V=150.0 PL=0  +MOVJ EC00514
ARCON
SMOVL C00515 BC00515 V=9.2  +MOVJ EC00515
SMOVL C00516 BC00516 V=9.2  +MOVJ EC00516
SMOVL C00517 BC00517 V=9.2  +MOVJ EC00517
ARCOF
SMOVL C00518 BC00518 V=800.0  +MOVJ EC00518
SMOVL C00519 BC00519 V=1000.0  +MOVJ EC00519
SFTOF3D
'EndPath W4121
'brak dostepu offset 5mm
MOVJ C00520 BC00520 VJ=100.00  +MOVJ EC00520 VJ=100.00
'Path W4122
SFTOF3D
SFTON3D P028
MOVJ C00521 BC00521 VJ=100.00  +MOVJ EC00521 VJ=100.00
SMOVL C00522 BC00522 V=800.0  +MOVJ EC00522
SMOVL C00523 BC00523 V=166.7 PL=0  +MOVJ EC00523
ARCON
SMOVL C00524 BC00524 V=11.7  +MOVJ EC00524
ARCOF
SMOVL C00525 BC00525 V=800.0  +MOVJ EC00525
SMOVL C00526 BC00526 V=1000.0  +MOVJ EC00526
SFTOF3D
'EndPath W4122
MOVJ C00527 BC00527 VJ=100.00  +MOVJ EC00527 VJ=100.00
'13
MOVJ C00528 BC00528 VJ=100.00  +MOVJ EC00528 VJ=100.00
'Path W4123
SFTOF3D
SFTON3D P030
MOVJ C00529 BC00529 VJ=100.00  +MOVJ EC00529 VJ=100.00
SMOVL C00530 BC00530 V=800.0  +MOVJ EC00530
SMOVL C00531 BC00531 V=150.0 PL=0  +MOVJ EC00531
MACRO1 MJ#(0) ARGF9
ARCON
SFTON3D P031
SMOVL C00532 BC00532 V=10.8  +MOVJ EC00532
ARCOF
SMOVL C00533 BC00533 V=800.0  +MOVJ EC00533
SMOVL C00534 BC00534 V=1000.0  +MOVJ EC00534
SFTOF3D
'EndPath W4123
'14
'15-brak
'Path W4212
SFTOF3D
SFTON3D P052
MOVJ C00535 BC00535 VJ=100.00  +MOVJ EC00535 VJ=100.00
SMOVL C00536 BC00536 V=800.0  +MOVJ EC00536
SMOVL C00537 BC00537 V=150.0 PL=0  +MOVJ EC00537
ARCON
SMOVL C00538 BC00538 V=10.8  +MOVJ EC00538
SMOVL C00539 BC00539 V=10.8  +MOVJ EC00539
SMOVL C00540 BC00540 V=10.8  +MOVJ EC00540
ARCOF
SMOVL C00541 BC00541 V=800.0  +MOVJ EC00541
MACRO1 MJ#(0) ARGF6
SMOVL C00542 BC00542 V=333.3  +MOVJ EC00542
SFTOF3D
'DODAC SHIFT
SFTON3D P088
SMOVL C00543 BC00543 V=133.3  +MOVJ EC00543
ARCON
SMOVL C00544 BC00544 V=10.8  +MOVJ EC00544
ARCOF
SMOVL C00545 BC00545 V=250.0  +MOVJ EC00545
SMOVL C00546 BC00546 V=1000.0  +MOVJ EC00546
SFTOF3D
'EndPath W4212
'16
'Path W4213
SFTOF3D
SFTON3D P053
MOVJ C00547 BC00547 VJ=100.00  +MOVJ EC00547 VJ=100.00
SMOVL C00548 BC00548 V=800.0  +MOVJ EC00548
SMOVL C00549 BC00549 V=150.0 PL=0  +MOVJ EC00549
MACRO1 MJ#(0) ARGF9
ARCON
SMOVL C00550 BC00550 V=10.8  +MOVJ EC00550
SMOVL C00551 BC00551 V=10.8  +MOVJ EC00551
SMOVL C00552 BC00552 V=10.8  +MOVJ EC00552
ARCOF
SMOVL C00553 BC00553 V=800.0  +MOVJ EC00553
SMOVL C00554 BC00554 V=1000.0  +MOVJ EC00554
SFTOF3D
'EndPath W4213
'Path W4124
SFTOF3D
SFTON3D P029
MOVJ C00555 BC00555 VJ=100.00  +MOVJ EC00555 VJ=100.00
SMOVL C00556 BC00556 V=800.0  +MOVJ EC00556
SMOVL C00557 BC00557 V=166.7 PL=0  +MOVJ EC00557
MACRO1 MJ#(0) ARGF14
ARCON
SMOVL C00558 BC00558 V=10.0  +MOVJ EC00558
SMOVL C00559 BC00559 V=10.0  +MOVJ EC00559
ARCOF
SMOVL C00560 BC00560 V=800.0  +MOVJ EC00560
SMOVL C00561 BC00561 V=1000.0  +MOVJ EC00561
SFTOF3D
'EndPath W4124
MOVJ C00562 BC00562 VJ=100.00  +MOVJ EC00562 VJ=100.00
'Path W4125
SFTOF3D
SFTON3D P029
MOVJ C00563 BC00563 VJ=100.00  +MOVJ EC00563 VJ=100.00
SMOVL C00564 BC00564 V=800.0  +MOVJ EC00564
SMOVL C00565 BC00565 V=150.0 PL=0  +MOVJ EC00565
ARCON
SMOVL C00566 BC00566 V=11.7  +MOVJ EC00566
SMOVL C00567 BC00567 V=11.7  +MOVJ EC00567
SMOVL C00568 BC00568 V=11.7  +MOVJ EC00568
ARCOF
SMOVL C00569 BC00569 V=800.0  +MOVJ EC00569
SMOVL C00570 BC00570 V=1000.0  +MOVJ EC00570
SFTOF3D
'EndPath W4125
MOVJ C00571 BC00571 VJ=100.00  +MOVJ EC00571 VJ=100.00
'Path W4126
SFTOF3D
SFTON3D P029
MOVJ C00572 BC00572 VJ=100.00  +MOVJ EC00572 VJ=100.00
SMOVL C00573 BC00573 V=800.0  +MOVJ EC00573
SMOVL C00574 BC00574 V=166.7 PL=0  +MOVJ EC00574
ARCON
SMOVL C00575 BC00575 V=11.7  +MOVJ EC00575
ARCON
SMOVL C00576 BC00576 V=11.7  +MOVJ EC00576
SMOVL C00577 BC00577 V=11.7  +MOVJ EC00577
ARCOF
SMOVL C00578 BC00578 V=800.0  +MOVJ EC00578
SMOVL C00579 BC00579 V=1000.0  +MOVJ EC00579
SFTOF3D
SFTON3D P080
MOVJ C00580 BC00580 VJ=100.00  +MOVJ EC00580 VJ=100.00
SMOVL C00581 BC00581 V=800.0  +MOVJ EC00581
SMOVL C00582 BC00582 V=166.7 PL=0  +MOVJ EC00582
MACRO1 MJ#(0) ARGF14
ARCON
SMOVL C00583 BC00583 V=10.0  +MOVJ EC00583
SMOVL C00584 BC00584 V=10.0  +MOVJ EC00584
ARCOF
SMOVL C00585 BC00585 V=800.0  +MOVJ EC00585
SMOVL C00586 BC00586 V=1000.0  +MOVJ EC00586
SFTOF3D
'EndPath W4124
MOVJ C00587 BC00587 VJ=100.00  +MOVJ EC00587 VJ=100.00
'Path W4125
SFTOF3D
SFTON3D P080
MOVJ C00588 BC00588 VJ=100.00  +MOVJ EC00588 VJ=100.00
SMOVL C00589 BC00589 V=800.0  +MOVJ EC00589
SMOVL C00590 BC00590 V=150.0 PL=0  +MOVJ EC00590
ARCON
SMOVL C00591 BC00591 V=11.7  +MOVJ EC00591
SMOVL C00592 BC00592 V=11.7  +MOVJ EC00592
SMOVL C00593 BC00593 V=11.7  +MOVJ EC00593
ARCOF
SMOVL C00594 BC00594 V=800.0  +MOVJ EC00594
SMOVL C00595 BC00595 V=1000.0  +MOVJ EC00595
SFTOF3D
'EndPath W4125
MOVJ C00596 BC00596 VJ=100.00  +MOVJ EC00596 VJ=100.00
'Path W4126
SFTOF3D
SFTON3D P080
MOVJ C00597 BC00597 VJ=100.00  +MOVJ EC00597 VJ=100.00
SMOVL C00598 BC00598 V=800.0  +MOVJ EC00598
SMOVL C00599 BC00599 V=166.7 PL=0  +MOVJ EC00599
ARCON
SMOVL C00600 BC00600 V=11.7  +MOVJ EC00600
ARCON
SMOVL C00601 BC00601 V=11.7  +MOVJ EC00601
SMOVL C00602 BC00602 V=11.7  +MOVJ EC00602
ARCOF
SMOVL C00603 BC00603 V=800.0  +MOVJ EC00603
SMOVL C00604 BC00604 V=1000.0  +MOVJ EC00604
SFTOF3D
'EndPath W4126
MOVJ C00605 BC00605 VJ=100.00  +MOVJ EC00605 VJ=100.00
'17
'Path W4127
SFTOF3D
SFTON3D P027
MOVJ C00606 BC00606 VJ=100.00  +MOVJ EC00606 VJ=100.00
SMOVL C00607 BC00607 V=800.0  +MOVJ EC00607
SMOVL C00608 BC00608 V=150.0 PL=0  +MOVJ EC00608
ARCON
SMOVL C00609 BC00609 V=10.0  +MOVJ EC00609
ARCOF
SMOVL C00610 BC00610 V=800.0  +MOVJ EC00610
SMOVL C00611 BC00611 V=1000.0  +MOVJ EC00611
SFTOF3D
'EndPath W4127
'Path W4128
SFTOF3D
SFTON3D P027
MOVJ C00612 BC00612 VJ=100.00  +MOVJ EC00612 VJ=100.00
SMOVL C00613 BC00613 V=800.0  +MOVJ EC00613
SMOVL C00614 BC00614 V=150.0 PL=0  +MOVJ EC00614
ARCON
SMOVL C00615 BC00615 V=11.7  +MOVJ EC00615
ARCOF
SMOVL C00616 BC00616 V=800.0  +MOVJ EC00616
SMOVL C00617 BC00617 V=1000.0  +MOVJ EC00617
SFTOF3D
'EndPath W4128
'Path W4129
SFTOF3D
SFTON3D P027
MOVJ C00618 BC00618 VJ=100.00  +MOVJ EC00618 VJ=100.00
SMOVL C00619 BC00619 V=800.0  +MOVJ EC00619
SMOVL C00620 BC00620 V=150.0 PL=0  +MOVJ EC00620
SMOVL C00621 BC00621 V=16.7  +MOVJ EC00621
ARCOF
SMOVL C00622 BC00622 V=800.0  +MOVJ EC00622
SMOVL C00623 BC00623 V=1000.0  +MOVJ EC00623
SFTOF3D
'EndPath W4129
'18
MOVJ C00624 BC00624 VJ=100.00  +MOVJ EC00624 VJ=100.00
'Path W4130
SFTOF3D
SFTON3D P024
MOVJ C00625 BC00625 VJ=100.00  +MOVJ EC00625 VJ=100.00
SMOVL C00626 BC00626 V=800.0  +MOVJ EC00626
SMOVL C00627 BC00627 V=150.0 PL=0  +MOVJ EC00627
ARCON
SMOVL C00628 BC00628 V=9.2  +MOVJ EC00628
SMOVL C00629 BC00629 V=9.2  +MOVJ EC00629
SMOVL C00630 BC00630 V=9.2  +MOVJ EC00630
SMOVL C00631 BC00631 V=9.2  +MOVJ EC00631
ARCOF
SMOVL C00632 BC00632 V=800.0  +MOVJ EC00632
SMOVL C00633 BC00633 V=1000.0  +MOVJ EC00633
SFTOF3D
'EndPath W4130
'Path W4860
SFTOF3D
SFTON3D P071
MOVJ C00634 BC00634 VJ=100.00  +MOVJ EC00634 VJ=100.00
SMOVL C00635 BC00635 V=800.0  +MOVJ EC00635
SMOVL C00636 BC00636 V=150.0 PL=0  +MOVJ EC00636
MACRO1 MJ#(0) ARGF9
ARCON
SMOVL C00637 BC00637 V=9.2  +MOVJ EC00637
SFTON3D P072
ARCON
SMOVL C00638 BC00638 V=9.2  +MOVJ EC00638
SMOVL C00639 BC00639 V=9.2  +MOVJ EC00639
ARCOF
SMOVL C00640 BC00640 V=333.3  +MOVJ EC00640
SMOVL C00641 BC00641 V=666.7  +MOVJ EC00641
SMOVL C00642 BC00642 V=333.3  +MOVJ EC00642
SMOVL C00643 BC00643 V=166.7 PL=0  +MOVJ EC00643
ARCON
SMOVL C00644 BC00644 V=9.2  +MOVJ EC00644
SMOVL C00645 BC00645 V=9.2  +MOVJ EC00645
ARCOF
SMOVL C00646 BC00646 V=800.0  +MOVJ EC00646
SMOVL C00647 BC00647 V=1000.0  +MOVJ EC00647
SFTOF3D
'EndPath W4860
'19
MOVJ C00648 BC00648 VJ=100.00  +MOVJ EC00648 VJ=100.00
'Path W4131
SFTOF3D
SFTON3D P023
MOVJ C00649 BC00649 VJ=100.00  +MOVJ EC00649 VJ=100.00
SMOVL C00650 BC00650 V=800.0  +MOVJ EC00650
SMOVL C00651 BC00651 V=166.7 PL=0  +MOVJ EC00651
MACRO1 MJ#(0) ARGF6
ARCON
SWVON WEV#(66)
SMOVL C00652 BC00652 V=7.5  +MOVJ EC00652
SMOVL C00653 BC00653 V=7.5  +MOVJ EC00653
SMOVL C00654 BC00654 V=7.5  +MOVJ EC00654
ARCOF
SWVOF
SMOVL C00655 BC00655 V=800.0  +MOVJ EC00655
SMOVL C00656 BC00656 V=1000.0  +MOVJ EC00656
SFTOF3D
'EndPath W4131
MOVJ C00657 BC00657 VJ=100.00  +MOVJ EC00657 VJ=100.00
'Path W4214
SFTOF3D
SFTON3D P089
MOVJ C00658 BC00658 VJ=100.00  +MOVJ EC00658 VJ=100.00
SMOVL C00659 BC00659 V=800.0  +MOVJ EC00659
SMOVL C00660 BC00660 V=150.0 PL=0  +MOVJ EC00660
MACRO1 MJ#(0) ARGF9
ARCON
SMOVL C00661 BC00661 V=9.2  +MOVJ EC00661
SFTON3D P050
SMOVL C00662 BC00662 V=9.2  +MOVJ EC00662
SMOVL C00663 BC00663 V=9.2  +MOVJ EC00663
ARCOF
SMOVL C00664 BC00664 V=800.0  +MOVJ EC00664
SMOVL C00665 BC00665 V=1000.0  +MOVJ EC00665
SFTOF3D
'EndPath W4214
'Path W4215
SFTOF3D
SFTON3D P051
MOVJ C00666 BC00666 VJ=100.00  +MOVJ EC00666 VJ=100.00
SMOVL C00667 BC00667 V=800.0  +MOVJ EC00667
SMOVL C00668 BC00668 V=150.0 PL=0  +MOVJ EC00668
MACRO1 MJ#(0) ARGF14
ARCON
SMOVL C00669 BC00669 V=9.2  +MOVJ EC00669
SMOVL C00670 BC00670 V=9.2  +MOVJ EC00670
SMOVL C00671 BC00671 V=9.2  +MOVJ EC00671
ARCOF
SMOVL C00672 BC00672 V=800.0  +MOVJ EC00672
SMOVL C00673 BC00673 V=1000.0  +MOVJ EC00673
SFTOF3D
'EndPath W4215
MOVJ C00674 BC00674 VJ=100.00  +MOVJ EC00674 VJ=100.00
'20
'offset 5mm
MOVJ C00675 BC00675 VJ=100.00  +MOVJ EC00675 VJ=100.00
MOVJ C00676 BC00676 VJ=100.00  +MOVJ EC00676 VJ=100.00
'Path W4132
SFTOF3D
SFTON3D P032
MOVJ C00677 BC00677 VJ=100.00  +MOVJ EC00677 VJ=100.00
SMOVL C00678 BC00678 V=800.0  +MOVJ EC00678
SMOVL C00679 BC00679 V=150.0 PL=0  +MOVJ EC00679
ARCON
SMOVL C00680 BC00680 V=10.0  +MOVJ EC00680
SMOVL C00681 BC00681 V=10.0  +MOVJ EC00681
ARCOF
SMOVL C00682 BC00682 V=800.0  +MOVJ EC00682
SMOVL C00683 BC00683 V=1000.0  +MOVJ EC00683
SFTOF3D
JUMP *FFF
'EndPath W4132
'Path W4133
SFTOF3D
SFTON3D P032
MOVJ C00684 BC00684 VJ=100.00  +MOVJ EC00684 VJ=100.00
SMOVL C00685 BC00685 V=800.0  +MOVJ EC00685
SMOVL C00686 BC00686 V=166.7 PL=0  +MOVJ EC00686
ARCON
SMOVL C00687 BC00687 V=10.0  +MOVJ EC00687
ARCOF
SMOVL C00688 BC00688 V=800.0  +MOVJ EC00688
SMOVL C00689 BC00689 V=1000.0  +MOVJ EC00689
SFTOF3D
'EndPath W4133
'Path W4134
SFTOF3D
SFTON3D P032
MOVJ C00690 BC00690 VJ=100.00  +MOVJ EC00690 VJ=100.00
SMOVL C00691 BC00691 V=800.0  +MOVJ EC00691
SMOVL C00692 BC00692 V=150.0 PL=0  +MOVJ EC00692
ARCON
SMOVL C00693 BC00693 V=10.0  +MOVJ EC00693
ARCOF
SMOVL C00694 BC00694 V=800.0  +MOVJ EC00694
*FFF
SMOVL C00695 BC00695 V=1000.0  +MOVJ EC00695
SFTOF3D
'EndPath W4134
'offset 5mm
MOVJ C00696 BC00696 VJ=100.00  +MOVJ EC00696 VJ=100.00
'Path W4135
SFTOF3D
SFTON3D P032
MOVJ C00697 BC00697 VJ=100.00  +MOVJ EC00697 VJ=100.00
SMOVL C00698 BC00698 V=800.0  +MOVJ EC00698
SMOVL C00699 BC00699 V=166.7 PL=0  +MOVJ EC00699
ARCON
SMOVL C00700 BC00700 V=10.0  +MOVJ EC00700
ARCOF
SMOVL C00701 BC00701 V=800.0  +MOVJ EC00701
SMOVL C00702 BC00702 V=1000.0  +MOVJ EC00702
SFTOF3D
'EndPath W4135
MOVJ C00703 BC00703 VJ=100.00  +MOVJ EC00703 VJ=100.00
'Path W4136
SFTOF3D
SFTON3D P032
MOVJ C00704 BC00704 VJ=100.00  +MOVJ EC00704 VJ=100.00
SMOVL C00705 BC00705 V=800.0  +MOVJ EC00705
SMOVL C00706 BC00706 V=166.7 PL=0  +MOVJ EC00706
ARCON
SMOVL C00707 BC00707 V=11.7  +MOVJ EC00707
SMOVL C00708 BC00708 V=11.7  +MOVJ EC00708
ARCOF
SMOVL C00709 BC00709 V=800.0  +MOVJ EC00709
SMOVL C00710 BC00710 V=1000.0  +MOVJ EC00710
SFTOF3D
'EndPath W4136
MOVJ C00711 BC00711 VJ=100.00  +MOVJ EC00711 VJ=100.00
MOVJ C00712 BC00712 VJ=100.00  +MOVJ EC00712 VJ=100.00
'Path W4137
SFTOF3D
SFTON3D P021
MOVJ C00713 BC00713 VJ=100.00  +MOVJ EC00713 VJ=100.00
SMOVL C00714 BC00714 V=800.0  +MOVJ EC00714
SMOVL C00715 BC00715 V=150.0 PL=0  +MOVJ EC00715
MACRO1 MJ#(0) ARGF9
ARCON
SFTON3D P022
SMOVL C00716 BC00716 V=10.0  +MOVJ EC00716
ARCOF
SMOVL C00717 BC00717 V=800.0  +MOVJ EC00717
SMOVL C00718 BC00718 V=1000.0  +MOVJ EC00718
SFTOF3D
'EndPath W4137
MOVJ C00719 BC00719 VJ=100.00  +MOVJ EC00719 VJ=100.00
'Path W4724
SFTOF3D
SFTON3D P095
MOVJ C00720 BC00720 VJ=100.00  +MOVJ EC00720 VJ=100.00
SMOVL C00721 BC00721 V=800.0  +MOVJ EC00721
SMOVL C00722 BC00722 V=150.0 PL=0  +MOVJ EC00722
ARCON
SMOVL C00723 BC00723 V=10.0  +MOVJ EC00723
SMOVL C00724 BC00724 V=10.0  +MOVJ EC00724
SMOVL C00725 BC00725 V=10.0  +MOVJ EC00725
ARCOF
SMOVL C00726 BC00726 V=800.0  +MOVJ EC00726
SMOVL C00727 BC00727 V=1000.0  +MOVJ EC00727
SFTOF3D
'EndPath W4724
'Path W4725
SFTOF3D
SFTON3D P096
MOVJ C00728 BC00728 VJ=100.00  +MOVJ EC00728 VJ=100.00
SMOVL C00729 BC00729 V=800.0  +MOVJ EC00729
SMOVL C00730 BC00730 V=150.0 PL=0  +MOVJ EC00730
ARCON
SMOVL C00731 BC00731 V=10.0  +MOVJ EC00731
SMOVL C00732 BC00732 V=10.0  +MOVJ EC00732
ARCOF
SMOVL C00733 BC00733 V=800.0  +MOVJ EC00733
SMOVL C00734 BC00734 V=1000.0  +MOVJ EC00734
SFTOF3D
'EndPath W4725
MOVJ C00735 BC00735 VJ=100.00  +MOVJ EC00735 VJ=100.00
'Path W4861
SFTOF3D
SFTON3D P071
MOVJ C00736 BC00736 VJ=100.00  +MOVJ EC00736 VJ=100.00
SMOVL C00737 BC00737 V=800.0  +MOVJ EC00737
SMOVL C00738 BC00738 V=150.0 PL=0  +MOVJ EC00738
MACRO1 MJ#(0) ARGF14
ARCON
SMOVL C00739 BC00739 V=9.2  +MOVJ EC00739
SFTON3D P073
SMOVL C00740 BC00740 V=9.2  +MOVJ EC00740
SMOVL C00741 BC00741 V=9.2  +MOVJ EC00741
ARCOF
SMOVL C00742 BC00742 V=800.0  +MOVJ EC00742
SMOVL C00743 BC00743 V=1000.0  +MOVJ EC00743
SFTOF3D
SMOVL C00744 BC00744 V=1000.0  +MOVJ EC00744
SFTOF3D
SFTON3D P080
MOVJ C00745 BC00745 VJ=100.00  +MOVJ EC00745 VJ=100.00
SMOVL C00746 BC00746 V=800.0  +MOVJ EC00746
SMOVL C00747 BC00747 V=150.0 PL=0  +MOVJ EC00747
MACRO1 MJ#(0) ARGF14
ARCON
SMOVL C00748 BC00748 V=9.2  +MOVJ EC00748
SFTON3D P080
SMOVL C00749 BC00749 V=9.2  +MOVJ EC00749
SMOVL C00750 BC00750 V=9.2  +MOVJ EC00750
ARCOF
SMOVL C00751 BC00751 V=800.0  +MOVJ EC00751
SMOVL C00752 BC00752 V=1000.0  +MOVJ EC00752
SFTOF3D
'EndPath W4861
MOVJ C00753 BC00753 VJ=100.00  +MOVJ EC00753 VJ=100.00
MOVJ C00754 BC00754 VJ=100.00  +MOVJ EC00754 VJ=100.00
MOVJ C00755 BC00755 VJ=100.00  +MOVJ EC00755 VJ=100.00
MOVJ C00756 BC00756 VJ=100.00  +MOVJ EC00756 VJ=100.00
MOVJ C00757 BC00757 VJ=100.00  +MOVJ EC00757 VJ=100.00
MOVJ C00758 BC00758 VJ=100.00  +MOVJ EC00758 VJ=100.00
MOVL C00759 BC00759 V=1000.0  +MOVJ EC00759 VJ=100.00
SFTON3D P081
MOVL C00760 BC00760 V=166.7 PL=0  +MOVJ EC00760 VJ=100.00
ARCON
SMOVL C00761 BC00761 V=9.2  +MOVJ EC00761
SMOVL C00762 BC00762 V=9.2  +MOVJ EC00762
SMOVL C00763 BC00763 V=9.2  +MOVJ EC00763
ARCOF
MOVL C00764 BC00764 V=666.7  +MOVJ EC00764 VJ=100.00
SFTOF3D
MOVJ C00765 BC00765 VJ=100.00  +MOVJ EC00765 VJ=100.00
CALL JOB:CLEAN-R1_KM_NEW
'cut_wire_dol
'cut_wire_dol
'cut_wire_dol
MOVJ C00766 BC00766 VJ=100.00  +MOVJ EC00766 VJ=100.00
MOVJ C00767 BC00767 VJ=100.00  +MOVJ EC00767 VJ=100.00
MOVJ C00768 BC00768 VJ=100.00  +MOVJ EC00768 VJ=100.00
'Path S4138
SFTOF3D
MOVJ C00769 BC00769 VJ=100.00  +MOVJ EC00769 VJ=100.00
MOVL C00770 BC00770 V=800.0  +MOVJ EC00770 VJ=100.00
SMOVL C00771 BC00771 V=166.7  +MOVJ EC00771
SREFP 3 C00772 BC00772  +REFP EC00772
CALL JOB:SEARCH-R1-S13D
SET P049 P006
SFTON3D P049
SMOVL C00773 BC00773 V=166.7  +MOVJ EC00773
SMOVL C00774 BC00774 V=166.7  +MOVJ EC00774
SREFP 3 C00775 BC00775  +REFP EC00775
CALL JOB:SEARCH-R1-S13D
SET P049 P006
SFTON3D P049
SMOVL C00776 BC00776 V=166.7  +MOVJ EC00776
MOVL C00777 BC00777 V=800.0  +MOVJ EC00777 VJ=100.00
MOVL C00778 BC00778 V=1000.0  +MOVJ EC00778 VJ=100.00
'EndPath S4138
'Path S4139
SFTOF3D
MOVJ C00779 BC00779 VJ=100.00  +MOVJ EC00779 VJ=100.00
MOVL C00780 BC00780 V=800.0  +MOVJ EC00780 VJ=100.00
SMOVL C00781 BC00781 V=166.7  +MOVJ EC00781
SREFP 3 C00782 BC00782  +REFP EC00782
CALL JOB:SEARCH-R1-S13D
SET P048 P006
SFTON3D P048
SMOVL C00783 BC00783 V=166.7  +MOVJ EC00783
SMOVL C00784 BC00784 V=166.7  +MOVJ EC00784
SREFP 3 C00785 BC00785  +REFP EC00785
CALL JOB:SEARCH-R1-S13D
SET P048 P006
SFTON3D P048
SMOVL C00786 BC00786 V=166.7  +MOVJ EC00786
MOVL C00787 BC00787 V=800.0  +MOVJ EC00787 VJ=100.00
MOVL C00788 BC00788 V=1000.0  +MOVJ EC00788 VJ=100.00
'EndPath S4139
'Path S4140
SFTOF3D
MOVJ C00789 BC00789 VJ=100.00  +MOVJ EC00789 VJ=100.00
MOVL C00790 BC00790 V=800.0  +MOVJ EC00790 VJ=100.00
SMOVL C00791 BC00791 V=166.7  +MOVJ EC00791
SREFP 3 C00792 BC00792  +REFP EC00792
CALL JOB:SEARCH-R1-S13D
SET P047 P006
SFTON3D P047
SMOVL C00793 BC00793 V=166.7  +MOVJ EC00793
SMOVL C00794 BC00794 V=166.7  +MOVJ EC00794
SREFP 3 C00795 BC00795  +REFP EC00795
CALL JOB:SEARCH-R1-S13D
SET P047 P006
SFTON3D P047
SMOVL C00796 BC00796 V=166.7  +MOVJ EC00796
MOVL C00797 BC00797 V=800.0  +MOVJ EC00797 VJ=100.00
MOVL C00798 BC00798 V=1000.0  +MOVJ EC00798 VJ=100.00
'EndPath S4140
MOVJ C00799 BC00799 VJ=100.00  +MOVJ EC00799 VJ=100.00
MOVJ C00800 BC00800 VJ=100.00  +MOVJ EC00800 VJ=100.00
MOVJ C00801 BC00801 VJ=100.00  +MOVJ EC00801 VJ=100.00
MOVJ C00802 BC00802 VJ=100.00  +MOVJ EC00802 VJ=100.00
'Path S4141
SFTOF3D
MOVJ C00803 BC00803 VJ=100.00  +MOVJ EC00803 VJ=100.00
MOVL C00804 BC00804 V=800.0  +MOVJ EC00804 VJ=100.00
SMOVL C00805 BC00805 V=166.7  +MOVJ EC00805
SREFP 3 C00806 BC00806  +REFP EC00806
CALL JOB:SEARCH-R1-S13D
SET P046 P006
SFTON3D P046
SMOVL C00807 BC00807 V=166.7  +MOVJ EC00807
SMOVL C00808 BC00808 V=166.7  +MOVJ EC00808
SREFP 3 C00809 BC00809  +REFP EC00809
CALL JOB:SEARCH-R1-S13D
SET P046 P006
SFTON3D P046
SMOVL C00810 BC00810 V=166.7  +MOVJ EC00810
MOVL C00811 BC00811 V=1000.0  +MOVJ EC00811 VJ=100.00
'EndPath S4141
'Path S4142
SFTOF3D
MOVJ C00812 BC00812 VJ=100.00  +MOVJ EC00812 VJ=100.00
MOVL C00813 BC00813 V=800.0  +MOVJ EC00813 VJ=100.00
SMOVL C00814 BC00814 V=166.7  +MOVJ EC00814
SREFP 3 C00815 BC00815  +REFP EC00815
CALL JOB:SEARCH-R1-S13D
SET P045 P006
SFTON3D P045
SMOVL C00816 BC00816 V=166.7  +MOVJ EC00816
SMOVL C00817 BC00817 V=166.7  +MOVJ EC00817
SREFP 3 C00818 BC00818  +REFP EC00818
CALL JOB:SEARCH-R1-S13D
SET P045 P006
SFTON3D P045
SMOVL C00819 BC00819 V=166.7  +MOVJ EC00819
MOVL C00820 BC00820 V=1000.0  +MOVJ EC00820 VJ=100.00
'EndPath S4142
'Path S4143
SFTOF3D
MOVJ C00821 BC00821 VJ=100.00  +MOVJ EC00821 VJ=100.00
MOVL C00822 BC00822 V=800.0  +MOVJ EC00822 VJ=100.00
SMOVL C00823 BC00823 V=166.7  +MOVJ EC00823
SREFP 3 C00824 BC00824  +REFP EC00824
CALL JOB:SEARCH-R1-S13D
SET P044 P006
SFTON3D P044
SMOVL C00825 BC00825 V=166.7  +MOVJ EC00825
SMOVL C00826 BC00826 V=166.7  +MOVJ EC00826
SREFP 3 C00827 BC00827  +REFP EC00827
CALL JOB:SEARCH-R1-S13D
SET P044 P006
SFTON3D P044
SMOVL C00828 BC00828 V=166.7  +MOVJ EC00828
MOVL C00829 BC00829 V=1000.0  +MOVJ EC00829 VJ=100.00
'EndPath S4143
MOVJ C00830 BC00830 VJ=100.00  +MOVJ EC00830 VJ=100.00
MOVJ C00831 BC00831 VJ=100.00  +MOVJ EC00831 VJ=100.00
'Path S4144
SFTOF3D
MOVJ C00832 BC00832 VJ=100.00  +MOVJ EC00832 VJ=100.00
MOVL C00833 BC00833 V=800.0  +MOVJ EC00833 VJ=100.00
SMOVL C00834 BC00834 V=166.7  +MOVJ EC00834
SREFP 3 C00835 BC00835  +REFP EC00835
CALL JOB:SEARCH-R1-S13D
SET P043 P006
SFTON3D P043
SMOVL C00836 BC00836 V=166.7  +MOVJ EC00836
SMOVL C00837 BC00837 V=166.7  +MOVJ EC00837
SREFP 3 C00838 BC00838  +REFP EC00838
CALL JOB:SEARCH-R1-S13D
SET P043 P006
SFTON3D P043
SMOVL C00839 BC00839 V=166.7  +MOVJ EC00839
MOVL C00840 BC00840 V=1000.0  +MOVJ EC00840 VJ=100.00
'EndPath S4144
'Path S4145
SFTOF3D
MOVJ C00841 BC00841 VJ=100.00  +MOVJ EC00841 VJ=100.00
MOVL C00842 BC00842 V=800.0  +MOVJ EC00842 VJ=100.00
SMOVL C00843 BC00843 V=166.7  +MOVJ EC00843
SREFP 3 C00844 BC00844  +REFP EC00844
CALL JOB:SEARCH-R1-S13D
SET P042 P006
SFTON3D P042
SMOVL C00845 BC00845 V=166.7  +MOVJ EC00845
SMOVL C00846 BC00846 V=166.7  +MOVJ EC00846
SREFP 3 C00847 BC00847  +REFP EC00847
CALL JOB:SEARCH-R1-S13D
SET P042 P006
SFTON3D P042
SMOVL C00848 BC00848 V=166.7  +MOVJ EC00848
MOVL C00849 BC00849 V=1000.0  +MOVJ EC00849 VJ=100.00
'EndPath S4145
'Path S4146
SFTOF3D
MOVJ C00850 BC00850 VJ=100.00  +MOVJ EC00850 VJ=100.00
MOVL C00851 BC00851 V=666.7  +MOVJ EC00851 VJ=100.00
SMOVL C00852 BC00852 V=166.7  +MOVJ EC00852
SREFP 3 C00853 BC00853  +REFP EC00853
CALL JOB:SEARCH-R1-S13D
SET P041 P006
SFTON3D P041
SMOVL C00854 BC00854 V=250.0  +MOVJ EC00854
SMOVL C00855 BC00855 V=166.7  +MOVJ EC00855
SREFP 3 C00856 BC00856  +REFP EC00856
CALL JOB:SEARCH-R1-S13D
SET P041 P006
SFTON3D P041
SMOVL C00857 BC00857 V=166.7  +MOVJ EC00857
SMOVL C00858 BC00858 V=166.7  +MOVJ EC00858
SREFP 3 C00859 BC00859  +REFP EC00859
CALL JOB:SEARCH-R1-S13D
SET P041 P006
SFTON3D P041
SMOVL C00860 BC00860 V=166.7  +MOVJ EC00860
MOVL C00861 BC00861 V=1000.0  +MOVJ EC00861 VJ=100.00
'EndPath S4146
'Path S4147
SFTOF3D
MOVJ C00862 BC00862 VJ=100.00  +MOVJ EC00862 VJ=100.00
SMOVL C00863 BC00863 V=666.7  +MOVJ EC00863
SMOVL C00864 BC00864 V=166.7  +MOVJ EC00864
SREFP 3 C00865 BC00865  +REFP EC00865
CALL JOB:SEARCH-R1-S13D
SET P040 P006
SFTON3D P040
SMOVL C00866 BC00866 V=166.7  +MOVJ EC00866
SMOVL C00867 BC00867 V=800.0  +MOVJ EC00867
SMOVL C00868 BC00868 V=166.7  +MOVJ EC00868
SREFP 3 C00869 BC00869  +REFP EC00869
CALL JOB:SEARCH-R1-S13D
SET P040 P006
SFTON3D P040
SMOVL C00870 BC00870 V=166.7  +MOVJ EC00870
SMOVL C00871 BC00871 V=166.7  +MOVJ EC00871
SREFP 3 C00872 BC00872  +REFP EC00872
CALL JOB:SEARCH-R1-S13D
SET P040 P006
SFTON3D P040
SMOVL C00873 BC00873 V=166.7  +MOVJ EC00873
MOVL C00874 BC00874 V=1000.0  +MOVJ EC00874 VJ=100.00
'EndPath S4147
'Path W4148
SFTOF3D
SFTON3D P040
MOVJ C00875 BC00875 VJ=100.00  +MOVJ EC00875 VJ=100.00
SMOVL C00876 BC00876 V=800.0  +MOVJ EC00876
SMOVL C00877 BC00877 V=150.0 PL=0  +MOVJ EC00877
ARCON
SMOVL C00878 BC00878 V=10.0  +MOVJ EC00878
ARCOF
SMOVL C00879 BC00879 V=800.0  +MOVJ EC00879
SMOVL C00880 BC00880 V=1000.0  +MOVJ EC00880
SFTOF3D
'EndPath W4148
'Path W4149
SFTOF3D
SFTON3D P040
MOVJ C00881 BC00881 VJ=100.00  +MOVJ EC00881 VJ=100.00
SMOVL C00882 BC00882 V=800.0  +MOVJ EC00882
SMOVL C00883 BC00883 V=150.0 PL=0  +MOVJ EC00883
ARCON
SMOVL C00884 BC00884 V=11.7  +MOVJ EC00884
ARCOF
SMOVL C00885 BC00885 V=800.0  +MOVJ EC00885
SMOVL C00886 BC00886 V=1000.0  +MOVJ EC00886
SFTOF3D
'EndPath W4149
'Path W4150
SFTOF3D
SFTON3D P040
MOVJ C00887 BC00887 VJ=15.00  +MOVJ EC00887 VJ=15.00
MOVJ C00888 BC00888 VJ=100.00  +MOVJ EC00888 VJ=100.00
SMOVL C00889 BC00889 V=800.0  +MOVJ EC00889
SMOVL C00890 BC00890 V=150.0 PL=0  +MOVJ EC00890
ARCON
SMOVL C00891 BC00891 V=11.7  +MOVJ EC00891
ARCOF
SMOVL C00892 BC00892 V=800.0  +MOVJ EC00892
SMOVL C00893 BC00893 V=1000.0  +MOVJ EC00893
SFTOF3D
'EndPath W4150
'
MOVJ C00894 BC00894 VJ=100.00  +MOVJ EC00894 VJ=100.00
MOVJ C00895 BC00895 VJ=100.00  +MOVJ EC00895 VJ=100.00
'Path W4151
SFTOF3D
SFTON3D P045
MOVJ C00896 BC00896 VJ=100.00  +MOVJ EC00896 VJ=100.00
SMOVL C00897 BC00897 V=800.0  +MOVJ EC00897
SMOVL C00898 BC00898 V=150.0 PL=0  +MOVJ EC00898
MACRO1 MJ#(0) ARGF9
ARCON
SMOVL C00899 BC00899 V=11.7  +MOVJ EC00899
ARCOF
SMOVL C00900 BC00900 V=800.0  +MOVJ EC00900
SMOVL C00901 BC00901 V=1000.0  +MOVJ EC00901
SFTOF3D
'EndPath W4151
'Path W4152
SFTOF3D
SFTON3D P044
MOVJ C00902 BC00902 VJ=100.00  +MOVJ EC00902 VJ=100.00
SMOVL C00903 BC00903 V=800.0  +MOVJ EC00903
SMOVL C00904 BC00904 V=166.7 PL=0  +MOVJ EC00904
ARCON
SMOVL C00905 BC00905 V=11.7  +MOVJ EC00905
ARCOF
SMOVL C00906 BC00906 V=800.0  +MOVJ EC00906
SMOVL C00907 BC00907 V=1000.0  +MOVJ EC00907
SFTOF3D
'EndPath W4152
'Path W4153
SFTOF3D
SFTON3D P046
MOVJ C00908 BC00908 VJ=100.00  +MOVJ EC00908 VJ=100.00
SMOVL C00909 BC00909 V=800.0  +MOVJ EC00909
SMOVL C00910 BC00910 V=166.7 PL=0  +MOVJ EC00910
MACRO1 MJ#(0) ARGF14
ARCON
SMOVL C00911 BC00911 V=10.0  +MOVJ EC00911
SMOVL C00912 BC00912 V=10.0  +MOVJ EC00912
ARCOF
SMOVL C00913 BC00913 V=800.0  +MOVJ EC00913
SMOVL C00914 BC00914 V=1000.0  +MOVJ EC00914
SFTOF3D
'EndPath W4153
MOVJ C00915 BC00915 VJ=100.00  +MOVJ EC00915 VJ=100.00
MOVJ C00916 BC00916 VJ=100.00  +MOVJ EC00916 VJ=100.00
MOVJ C00917 BC00917 VJ=100.00  +MOVJ EC00917 VJ=100.00
MOVJ C00918 BC00918 VJ=100.00  +MOVJ EC00918 VJ=100.00
'1
'uwaga na podajnik
'Path W4154
SFTOF3D
SFTON3D P048
MOVJ C00919 BC00919 VJ=100.00  +MOVJ EC00919 VJ=100.00
SMOVL C00920 BC00920 V=800.0  +MOVJ EC00920
SMOVL C00921 BC00921 V=150.0 PL=0  +MOVJ EC00921
ARCON
SMOVL C00922 BC00922 V=10.0  +MOVJ EC00922
ARCOF
SMOVL C00923 BC00923 V=800.0  +MOVJ EC00923
SMOVL C00924 BC00924 V=1000.0  +MOVJ EC00924
SFTOF3D
'EndPath W4154
'Path W4155
SFTOF3D
SFTON3D P049
MOVJ C00925 BC00925 VJ=100.00  +MOVJ EC00925 VJ=100.00
SMOVL C00926 BC00926 V=800.0  +MOVJ EC00926
SMOVL C00927 BC00927 V=150.0 PL=0  +MOVJ EC00927
MACRO1 MJ#(0) ARGF6
ARCON
SMOVL C00928 BC00928 V=9.2  +MOVJ EC00928
SMOVL C00929 BC00929 V=9.2  +MOVJ EC00929
SMOVL C00930 BC00930 V=9.2  +MOVJ EC00930
SMOVL C00931 BC00931 V=9.2  +MOVJ EC00931
SMOVL C00932 BC00932 V=9.2  +MOVJ EC00932
ARCOF
SMOVL C00933 BC00933 V=800.0  +MOVJ EC00933
SMOVL C00934 BC00934 V=500.0  +MOVJ EC00934
SMOVL C00935 BC00935 V=133.3  +MOVJ EC00935
ARCON
SMOVL C00936 BC00936 V=13.3  +MOVJ EC00936
ARCOF
SMOVL C00937 BC00937 V=166.7  +MOVJ EC00937
ARCON
SMOVL C00938 BC00938 V=10.0  +MOVJ EC00938
ARCOF
SMOVL C00939 BC00939 V=250.0  +MOVJ EC00939
SMOVL C00940 BC00940 V=500.0  +MOVJ EC00940
SMOVL C00941 BC00941 V=500.0  +MOVJ EC00941
SMOVL C00942 BC00942 V=500.0  +MOVJ EC00942
SMOVL C00943 BC00943 V=133.3  +MOVJ EC00943
ARCON
SMOVL C00944 BC00944 V=13.3  +MOVJ EC00944
ARCOF
SMOVL C00945 BC00945 V=166.7  +MOVJ EC00945
SMOVL C00946 BC00946 V=166.7  +MOVJ EC00946
ARCON
SMOVL C00947 BC00947 V=10.0  +MOVJ EC00947
ARCOF
SMOVL C00948 BC00948 V=800.0  +MOVJ EC00948
SFTOF3D
'EndPath W4155
MOVJ C00949 BC00949 VJ=100.00  +MOVJ EC00949 VJ=100.00
MOVJ C00950 BC00950 VJ=100.00  +MOVJ EC00950 VJ=100.00
MOVJ C00951 BC00951 VJ=100.00  +MOVJ EC00951 VJ=100.00
MOVJ C00952 BC00952 VJ=100.00  +MOVJ EC00952 VJ=100.00
'2
'Path W4156
SFTOF3D
SFTON3D P043
MOVJ C00953 BC00953 VJ=100.00  +MOVJ EC00953 VJ=100.00
SMOVL C00954 BC00954 V=800.0  +MOVJ EC00954
SMOVL C00955 BC00955 V=166.7 PL=0  +MOVJ EC00955
MACRO1 MJ#(0) ARGF9
ARCON
SMOVL C00956 BC00956 V=11.7  +MOVJ EC00956
ARCOF
SMOVL C00957 BC00957 V=800.0  +MOVJ EC00957
SMOVL C00958 BC00958 V=1000.0  +MOVJ EC00958
SFTOF3D
'EndPath W4156
'Path W4157
SFTOF3D
SFTON3D P042
MOVJ C00959 BC00959 VJ=100.00  +MOVJ EC00959 VJ=100.00
SMOVL C00960 BC00960 V=800.0  +MOVJ EC00960
SMOVL C00961 BC00961 V=150.0 PL=0  +MOVJ EC00961
ARCON
SMOVL C00962 BC00962 V=11.7  +MOVJ EC00962
ARCOF
SMOVL C00963 BC00963 V=800.0  +MOVJ EC00963
SMOVL C00964 BC00964 V=1000.0  +MOVJ EC00964
SFTOF3D
'EndPath W4157
'3
MOVJ C00965 BC00965 VJ=100.00  +MOVJ EC00965 VJ=100.00
MOVJ C00966 BC00966 VJ=100.00  +MOVJ EC00966 VJ=100.00
MOVJ C00967 BC00967 VJ=100.00  +MOVJ EC00967 VJ=100.00
MOVJ C00968 BC00968 VJ=100.00  +MOVJ EC00968 VJ=100.00
'Path W4158
SFTOF3D
SFTON3D P047
MOVJ C00969 BC00969 VJ=100.00  +MOVJ EC00969 VJ=100.00
SMOVL C00970 BC00970 V=800.0  +MOVJ EC00970
SMOVL C00971 BC00971 V=150.0 PL=0  +MOVJ EC00971
ARCON
SMOVL C00972 BC00972 V=11.7  +MOVJ EC00972
ARCOF
SMOVL C00973 BC00973 V=800.0  +MOVJ EC00973
SMOVL C00974 BC00974 V=1000.0  +MOVJ EC00974
SFTOF3D
'EndPath W4158
'Path W4159
SFTOF3D
SFTON3D P047
MOVJ C00975 BC00975 VJ=100.00  +MOVJ EC00975 VJ=100.00
SMOVL C00976 BC00976 V=800.0  +MOVJ EC00976
SMOVL C00977 BC00977 V=150.0 PL=0  +MOVJ EC00977
ARCON
SMOVL C00978 BC00978 V=11.7  +MOVJ EC00978
ARCOF
SMOVL C00979 BC00979 V=800.0  +MOVJ EC00979
SMOVL C00980 BC00980 V=1000.0  +MOVJ EC00980
SFTOF3D
'EndPath W4159
MOVJ C00981 BC00981 VJ=100.00  +MOVJ EC00981 VJ=100.00
MOVJ C00982 BC00982 VJ=100.00  +MOVJ EC00982 VJ=100.00
MOVJ C00983 BC00983 VJ=100.00  +MOVJ EC00983 VJ=100.00
MOVJ C00984 BC00984 VJ=100.00  +MOVJ EC00984 VJ=100.00
'Path W4160
SFTOF3D
SFTON3D P043
MOVJ C00985 BC00985 VJ=100.00  +MOVJ EC00985 VJ=100.00
SMOVL C00986 BC00986 V=800.0  +MOVJ EC00986
SMOVL C00987 BC00987 V=150.0 PL=0  +MOVJ EC00987
ARCON
SMOVL C00988 BC00988 V=11.7  +MOVJ EC00988
ARCOF
SMOVL C00989 BC00989 V=800.0  +MOVJ EC00989
SMOVL C00990 BC00990 V=1000.0  +MOVJ EC00990
SFTOF3D
'EndPath W4160
'Path W4161
SFTOF3D
SFTON3D P042
MOVJ C00991 BC00991 VJ=100.00  +MOVJ EC00991 VJ=100.00
SMOVL C00992 BC00992 V=800.0  +MOVJ EC00992
SMOVL C00993 BC00993 V=166.7 PL=0  +MOVJ EC00993
ARCON
SMOVL C00994 BC00994 V=11.7  +MOVJ EC00994
ARCOF
SMOVL C00995 BC00995 V=800.0  +MOVJ EC00995
SMOVL C00996 BC00996 V=1000.0  +MOVJ EC00996
SFTOF3D
'EndPath W4161
MOVJ C00997 BC00997 VJ=100.00  +MOVJ EC00997 VJ=100.00
'Path W4162
SFTOF3D
SFTON3D P046
MOVJ C00998 BC00998 VJ=100.00  +MOVJ EC00998 VJ=100.00
SMOVL C00999 BC00999 V=800.0  +MOVJ EC00999
SMOVL C01000 BC01000 V=166.7 PL=0  +MOVJ EC01000
MACRO1 MJ#(0) ARGF14
ARCON
SMOVL C01001 BC01001 V=10.0  +MOVJ EC01001
ARCOF
SMOVL C01002 BC01002 V=800.0  +MOVJ EC01002
SMOVL C01003 BC01003 V=1000.0  +MOVJ EC01003
SFTOF3D
'EndPath W4162
'Path W4163
SFTOF3D
SFTON3D P044
MOVJ C01004 BC01004 VJ=100.00  +MOVJ EC01004 VJ=100.00
SMOVL C01005 BC01005 V=800.0  +MOVJ EC01005
SMOVL C01006 BC01006 V=150.0 PL=0  +MOVJ EC01006
MACRO1 MJ#(0) ARGF9
ARCON
SMOVL C01007 BC01007 V=11.7  +MOVJ EC01007
ARCOF
SMOVL C01008 BC01008 V=800.0  +MOVJ EC01008
SMOVL C01009 BC01009 V=1000.0  +MOVJ EC01009
SFTOF3D
'EndPath W4163
MOVJ C01010 BC01010 VJ=100.00  +MOVJ EC01010 VJ=100.00
'Path W4164
SFTOF3D
SFTON3D P041
MOVJ C01011 BC01011 VJ=100.00  +MOVJ EC01011 VJ=100.00
SMOVL C01012 BC01012 V=800.0  +MOVJ EC01012
SMOVL C01013 BC01013 V=150.0 PL=0  +MOVJ EC01013
MACRO1 MJ#(0) ARGF14
ARCON
SMOVL C01014 BC01014 V=10.0  +MOVJ EC01014
SMOVL C01015 BC01015 V=10.0  +MOVJ EC01015
SMOVL C01016 BC01016 V=10.0  +MOVJ EC01016
ARCOF
SMOVL C01017 BC01017 V=800.0  +MOVJ EC01017
SMOVL C01018 BC01018 V=1000.0  +MOVJ EC01018
SFTOF3D
'EndPath W4164
JUMP *L_1
'Path W4165
SFTOF3D
SFTON3D P041
MOVJ C01019 BC01019 VJ=100.00  +MOVJ EC01019 VJ=100.00
SMOVL C01020 BC01020 V=800.0  +MOVJ EC01020
SMOVL C01021 BC01021 V=150.0 PL=0  +MOVJ EC01021
SMOVL C01022 BC01022 V=10.0  +MOVJ EC01022
ARCOF
SMOVL C01023 BC01023 V=800.0  +MOVJ EC01023
SMOVL C01024 BC01024 V=1000.0  +MOVJ EC01024
SFTOF3D
'EndPath W4165
MOVJ C01025 BC01025 VJ=100.00  +MOVJ EC01025 VJ=100.00
'Path W4166
SFTOF3D
SFTON3D P041
MOVJ C01026 BC01026 VJ=100.00  +MOVJ EC01026 VJ=100.00
SMOVL C01027 BC01027 V=800.0  +MOVJ EC01027
SMOVL C01028 BC01028 V=150.0 PL=0  +MOVJ EC01028
SMOVL C01029 BC01029 V=10.0  +MOVJ EC01029
ARCOF
SMOVL C01030 BC01030 V=800.0  +MOVJ EC01030
SMOVL C01031 BC01031 V=1000.0  +MOVJ EC01031
SFTOF3D
'EndPath W4166
*L_1
MOVJ C01032 BC01032 VJ=100.00  +MOVJ EC01032 VJ=100.00
MOVJ C01033 BC01033 VJ=100.00  +MOVJ EC01033 VJ=100.00
MOVJ C01034 BC01034 VJ=100.00  +MOVJ EC01034 VJ=100.00
END
